//     PlcTask Inputs/GVL_iXlinker.EtherCAT_Master_EPPxxxx.Beckhoff_EPP3xxx.Beckhoff_EPP3xxxEK1122.A_0023_EPP3744_1041_0019.AI_Inputs_Channel_2.Value <-> AI Inputs Channel 2/Value
//     PlcTask Inputs/GVL_iXlinker.EtherCAT_Master_EPPxxxx.Beckhoff_EPP3xxx.Beckhoff_EPP3xxxEK1122.A_0023_EPP3744_1041_0019.AI_Inputs_Channel_3.Value <-> AI Inputs Channel 3/Value
//     PlcTask Inputs/GVL_iXlinker.EtherCAT_Master_EPPxxxx.Beckhoff_EPP3xxx.Beckhoff_EPP3xxxEK1122.A_0023_EPP3744_1041_0019.AI_Inputs_Channel_4.Value <-> AI Inputs Channel 4/Value
//     PlcTask Inputs/GVL_iXlinker.EtherCAT_Master_EPPxxxx.Beckhoff_EPP3xxx.Beckhoff_EPP3xxxEK1122.A_0023_EPP3744_1041_0019.DEV_Inputs_Device.Safe_State_Active <-> DEV Inputs Device/Safe State Active
//     PlcTask Inputs/GVL_iXlinker.EtherCAT_Master_EPPxxxx.Beckhoff_EPP3xxx.Beckhoff_EPP3xxxEK1122.A_0023_EPP3744_1041_0019.DEV_Inputs_Device.Sync_error <-> DEV Inputs Device/Sync error
//     PlcTask Inputs/GVL_iXlinker.EtherCAT_Master_EPPxxxx.Beckhoff_EPP3xxx.Beckhoff_EPP3xxxEK1122.A_0023_EPP3744_1041_0019.DEV_Inputs_Device.Undervoltage_Us <-> DEV Inputs Device/Undervoltage Us
//     PlcTask Inputs/GVL_iXlinker.EtherCAT_Master_EPPxxxx.Beckhoff_EPP3xxx.Beckhoff_EPP3xxxEK1122.A_0023_EPP3744_1041_0019.DEV_Inputs_Device.Undervoltage_Up <-> DEV Inputs Device/Undervoltage Up
//     PlcTask Inputs/GVL_iXlinker.EtherCAT_Master_EPPxxxx.Beckhoff_EPP3xxx.Beckhoff_EPP3xxxEK1122.A_0023_EPP3744_1041_0019.DEV_Inputs_Device.TxPDO_Toggle <-> DEV Inputs Device/TxPDO Toggle
//     PlcTask Outputs/GVL_iXlinker.EtherCAT_Master_EPPxxxx.Beckhoff_EPP3xxx.Beckhoff_EPP3xxxEK1122.A_0023_EPP3744_1041_0019.DIG_Outputs.Output[0] <-> DIG Outputs/Output 1
//     PlcTask Outputs/GVL_iXlinker.EtherCAT_Master_EPPxxxx.Beckhoff_EPP3xxx.Beckhoff_EPP3xxxEK1122.A_0023_EPP3744_1041_0019.DIG_Outputs.Output[1] <-> DIG Outputs/Output 2
//     PlcTask Outputs/GVL_iXlinker.EtherCAT_Master_EPPxxxx.Beckhoff_EPP3xxx.Beckhoff_EPP3xxxEK1122.A_0023_EPP3744_1041_0019.DEV_Outputs_Device.Set_safe_state <-> DEV Outputs Device/Set safe state
//     PlcTask Inputs/GVL_iXlinker.EtherCAT_Master_EPPxxxx.Beckhoff_EPP3xxx.Beckhoff_EPP3xxxEK1122.A_0023_EPP3744_1041_0019.WcState.WcState <-> WcState/WcState
//     PlcTask Inputs/GVL_iXlinker.EtherCAT_Master_EPPxxxx.Beckhoff_EPP3xxx.Beckhoff_EPP3xxxEK1122.A_0023_EPP3744_1041_0019.WcState.InputToggle <-> WcState/InputToggle
//     PlcTask Inputs/GVL_iXlinker.EtherCAT_Master_EPPxxxx.Beckhoff_EPP3xxx.Beckhoff_EPP3xxxEK1122.A_0023_EPP3744_1041_0019.InfoData.AdsAddr <-> InfoData/AdsAddr
//     PlcTask Inputs/GVL_iXlinker.EtherCAT_Master_EPPxxxx.Beckhoff_EPP3xxx.Beckhoff_EPP3xxxEK1122.A_0023_EPP3744_1041_0019.InfoData.State <-> InfoData/State
//   PLC/PLC Instance <-> EtherCAT Master EPPxxxx/Beckhoff EPP3xxx/Beckhoff EPP3xxxEK1122/A_0024(EPP3744-1041-0020)
//     PlcTask Inputs/GVL_iXlinker.EtherCAT_Master_EPPxxxx.Beckhoff_EPP3xxx.Beckhoff_EPP3xxxEK1122.A_0024_EPP3744_1041_0020.DIG_Inputs.Input[0] <-> DIG Inputs/Input 1
//     PlcTask Inputs/GVL_iXlinker.EtherCAT_Master_EPPxxxx.Beckhoff_EPP3xxx.Beckhoff_EPP3xxxEK1122.A_0024_EPP3744_1041_0020.DIG_Inputs.Input[1] <-> DIG Inputs/Input 2
//     PlcTask Inputs/GVL_iXlinker.EtherCAT_Master_EPPxxxx.Beckhoff_EPP3xxx.Beckhoff_EPP3xxxEK1122.A_0024_EPP3744_1041_0020.DIG_Inputs.Input[2] <-> DIG Inputs/Input 3
//     PlcTask Inputs/GVL_iXlinker.EtherCAT_Master_EPPxxxx.Beckhoff_EPP3xxx.Beckhoff_EPP3xxxEK1122.A_0024_EPP3744_1041_0020.DIG_Inputs.Input[3] <-> DIG Inputs/Input 4
//     PlcTask Inputs/GVL_iXlinker.EtherCAT_Master_EPPxxxx.Beckhoff_EPP3xxx.Beckhoff_EPP3xxxEK1122.A_0024_EPP3744_1041_0020.DIG_Inputs.Input[4] <-> DIG Inputs/Input 5
//     PlcTask Inputs/GVL_iXlinker.EtherCAT_Master_EPPxxxx.Beckhoff_EPP3xxx.Beckhoff_EPP3xxxEK1122.A_0024_EPP3744_1041_0020.DIG_Inputs.Input[5] <-> DIG Inputs/Input 6
//     PlcTask Inputs/GVL_iXlinker.EtherCAT_Master_EPPxxxx.Beckhoff_EPP3xxx.Beckhoff_EPP3xxxEK1122.A_0024_EPP3744_1041_0020.AI_Inputs_Channel_1.Status/Underrange <-> AI Inputs Channel 1/Status/Underrange
//     PlcTask Inputs/GVL_iXlinker.EtherCAT_Master_EPPxxxx.Beckhoff_EPP3xxx.Beckhoff_EPP3xxxEK1122.A_0024_EPP3744_1041_0020.AI_Inputs_Channel_2.Status/Underrange <-> AI Inputs Channel 2/Status/Underrange
//     PlcTask Inputs/GVL_iXlinker.EtherCAT_Master_EPPxxxx.Beckhoff_EPP3xxx.Beckhoff_EPP3xxxEK1122.A_0024_EPP3744_1041_0020.AI_Inputs_Channel_3.Status/Underrange <-> AI Inputs Channel 3/Status/Underrange
//     PlcTask Inputs/GVL_iXlinker.EtherCAT_Master_EPPxxxx.Beckhoff_EPP3xxx.Beckhoff_EPP3xxxEK1122.A_0024_EPP3744_1041_0020.AI_Inputs_Channel_4.Status/Underrange <-> AI Inputs Channel 4/Status/Underrange
//     PlcTask Inputs/GVL_iXlinker.EtherCAT_Master_EPPxxxx.Beckhoff_EPP3xxx.Beckhoff_EPP3xxxEK1122.A_0024_EPP3744_1041_0020.AI_Inputs_Channel_1.Status/Overrange <-> AI Inputs Channel 1/Status/Overrange
//     PlcTask Inputs/GVL_iXlinker.EtherCAT_Master_EPPxxxx.Beckhoff_EPP3xxx.Beckhoff_EPP3xxxEK1122.A_0024_EPP3744_1041_0020.AI_Inputs_Channel_2.Status/Overrange <-> AI Inputs Channel 2/Status/Overrange
//     PlcTask Inputs/GVL_iXlinker.EtherCAT_Master_EPPxxxx.Beckhoff_EPP3xxx.Beckhoff_EPP3xxxEK1122.A_0024_EPP3744_1041_0020.AI_Inputs_Channel_3.Status/Overrange <-> AI Inputs Channel 3/Status/Overrange
//     PlcTask Inputs/GVL_iXlinker.EtherCAT_Master_EPPxxxx.Beckhoff_EPP3xxx.Beckhoff_EPP3xxxEK1122.A_0024_EPP3744_1041_0020.AI_Inputs_Channel_4.Status/Overrange <-> AI Inputs Channel 4/Status/Overrange
//     PlcTask Inputs/GVL_iXlinker.EtherCAT_Master_EPPxxxx.Beckhoff_EPP3xxx.Beckhoff_EPP3xxxEK1122.A_0024_EPP3744_1041_0020.AI_Inputs_Channel_1.Status/Limit_1 <-> AI Inputs Channel 1/Status/Limit 1
//     PlcTask Inputs/GVL_iXlinker.EtherCAT_Master_EPPxxxx.Beckhoff_EPP3xxx.Beckhoff_EPP3xxxEK1122.A_0024_EPP3744_1041_0020.AI_Inputs_Channel_1.Status/Limit_2 <-> AI Inputs Channel 1/Status/Limit 2
//     PlcTask Inputs/GVL_iXlinker.EtherCAT_Master_EPPxxxx.Beckhoff_EPP3xxx.Beckhoff_EPP3xxxEK1122.A_0024_EPP3744_1041_0020.AI_Inputs_Channel_2.Status/Limit_1 <-> AI Inputs Channel 2/Status/Limit 1
//     PlcTask Inputs/GVL_iXlinker.EtherCAT_Master_EPPxxxx.Beckhoff_EPP3xxx.Beckhoff_EPP3xxxEK1122.A_0024_EPP3744_1041_0020.AI_Inputs_Channel_2.Status/Limit_2 <-> AI Inputs Channel 2/Status/Limit 2
//     PlcTask Inputs/GVL_iXlinker.EtherCAT_Master_EPPxxxx.Beckhoff_EPP3xxx.Beckhoff_EPP3xxxEK1122.A_0024_EPP3744_1041_0020.AI_Inputs_Channel_3.Status/Limit_1 <-> AI Inputs Channel 3/Status/Limit 1
//     PlcTask Inputs/GVL_iXlinker.EtherCAT_Master_EPPxxxx.Beckhoff_EPP3xxx.Beckhoff_EPP3xxxEK1122.A_0024_EPP3744_1041_0020.AI_Inputs_Channel_3.Status/Limit_2 <-> AI Inputs Channel 3/Status/Limit 2
//     PlcTask Inputs/GVL_iXlinker.EtherCAT_Master_EPPxxxx.Beckhoff_EPP3xxx.Beckhoff_EPP3xxxEK1122.A_0024_EPP3744_1041_0020.AI_Inputs_Channel_4.Status/Limit_1 <-> AI Inputs Channel 4/Status/Limit 1
//     PlcTask Inputs/GVL_iXlinker.EtherCAT_Master_EPPxxxx.Beckhoff_EPP3xxx.Beckhoff_EPP3xxxEK1122.A_0024_EPP3744_1041_0020.AI_Inputs_Channel_4.Status/Limit_2 <-> AI Inputs Channel 4/Status/Limit 2
//     PlcTask Inputs/GVL_iXlinker.EtherCAT_Master_EPPxxxx.Beckhoff_EPP3xxx.Beckhoff_EPP3xxxEK1122.A_0024_EPP3744_1041_0020.AI_Inputs_Channel_1.Status/Error <-> AI Inputs Channel 1/Status/Error
//     PlcTask Inputs/GVL_iXlinker.EtherCAT_Master_EPPxxxx.Beckhoff_EPP3xxx.Beckhoff_EPP3xxxEK1122.A_0024_EPP3744_1041_0020.AI_Inputs_Channel_2.Status/Error <-> AI Inputs Channel 2/Status/Error
//     PlcTask Inputs/GVL_iXlinker.EtherCAT_Master_EPPxxxx.Beckhoff_EPP3xxx.Beckhoff_EPP3xxxEK1122.A_0024_EPP3744_1041_0020.AI_Inputs_Channel_3.Status/Error <-> AI Inputs Channel 3/Status/Error
//     PlcTask Inputs/GVL_iXlinker.EtherCAT_Master_EPPxxxx.Beckhoff_EPP3xxx.Beckhoff_EPP3xxxEK1122.A_0024_EPP3744_1041_0020.AI_Inputs_Channel_4.Status/Error <-> AI Inputs Channel 4/Status/Error
//     PlcTask Inputs/GVL_iXlinker.EtherCAT_Master_EPPxxxx.Beckhoff_EPP3xxx.Beckhoff_EPP3xxxEK1122.A_0024_EPP3744_1041_0020.AI_Inputs_Channel_1.Status/TxPDO_State <-> AI Inputs Channel 1/Status/TxPDO State
//     PlcTask Inputs/GVL_iXlinker.EtherCAT_Master_EPPxxxx.Beckhoff_EPP3xxx.Beckhoff_EPP3xxxEK1122.A_0024_EPP3744_1041_0020.AI_Inputs_Channel_2.Status/TxPDO_State <-> AI Inputs Channel 2/Status/TxPDO State
//     PlcTask Inputs/GVL_iXlinker.EtherCAT_Master_EPPxxxx.Beckhoff_EPP3xxx.Beckhoff_EPP3xxxEK1122.A_0024_EPP3744_1041_0020.AI_Inputs_Channel_3.Status/TxPDO_State <-> AI Inputs Channel 3/Status/TxPDO State
//     PlcTask Inputs/GVL_iXlinker.EtherCAT_Master_EPPxxxx.Beckhoff_EPP3xxx.Beckhoff_EPP3xxxEK1122.A_0024_EPP3744_1041_0020.AI_Inputs_Channel_4.Status/TxPDO_State <-> AI Inputs Channel 4/Status/TxPDO State
//     PlcTask Inputs/GVL_iXlinker.EtherCAT_Master_EPPxxxx.Beckhoff_EPP3xxx.Beckhoff_EPP3xxxEK1122.A_0024_EPP3744_1041_0020.AI_Inputs_Channel_1.Status/TxPDO_Toggle <-> AI Inputs Channel 1/Status/TxPDO Toggle
//     PlcTask Inputs/GVL_iXlinker.EtherCAT_Master_EPPxxxx.Beckhoff_EPP3xxx.Beckhoff_EPP3xxxEK1122.A_0024_EPP3744_1041_0020.AI_Inputs_Channel_2.Status/TxPDO_Toggle <-> AI Inputs Channel 2/Status/TxPDO Toggle
//     PlcTask Inputs/GVL_iXlinker.EtherCAT_Master_EPPxxxx.Beckhoff_EPP3xxx.Beckhoff_EPP3xxxEK1122.A_0024_EPP3744_1041_0020.AI_Inputs_Channel_3.Status/TxPDO_Toggle <-> AI Inputs Channel 3/Status/TxPDO Toggle
//     PlcTask Inputs/GVL_iXlinker.EtherCAT_Master_EPPxxxx.Beckhoff_EPP3xxx.Beckhoff_EPP3xxxEK1122.A_0024_EPP3744_1041_0020.AI_Inputs_Channel_4.Status/TxPDO_Toggle <-> AI Inputs Channel 4/Status/TxPDO Toggle
//     PlcTask Inputs/GVL_iXlinker.EtherCAT_Master_EPPxxxx.Beckhoff_EPP3xxx.Beckhoff_EPP3xxxEK1122.A_0024_EPP3744_1041_0020.AI_Inputs_Channel_1.Value <-> AI Inputs Channel 1/Value
//     PlcTask Inputs/GVL_iXlinker.EtherCAT_Master_EPPxxxx.Beckhoff_EPP3xxx.Beckhoff_EPP3xxxEK1122.A_0024_EPP3744_1041_0020.AI_Inputs_Channel_2.Value <-> AI Inputs Channel 2/Value
//     PlcTask Inputs/GVL_iXlinker.EtherCAT_Master_EPPxxxx.Beckhoff_EPP3xxx.Beckhoff_EPP3xxxEK1122.A_0024_EPP3744_1041_0020.AI_Inputs_Channel_3.Value <-> AI Inputs Channel 3/Value
//     PlcTask Inputs/GVL_iXlinker.EtherCAT_Master_EPPxxxx.Beckhoff_EPP3xxx.Beckhoff_EPP3xxxEK1122.A_0024_EPP3744_1041_0020.AI_Inputs_Channel_4.Value <-> AI Inputs Channel 4/Value
//     PlcTask Inputs/GVL_iXlinker.EtherCAT_Master_EPPxxxx.Beckhoff_EPP3xxx.Beckhoff_EPP3xxxEK1122.A_0024_EPP3744_1041_0020.DEV_Inputs_Device.Safe_State_Active <-> DEV Inputs Device/Safe State Active
//     PlcTask Inputs/GVL_iXlinker.EtherCAT_Master_EPPxxxx.Beckhoff_EPP3xxx.Beckhoff_EPP3xxxEK1122.A_0024_EPP3744_1041_0020.DEV_Inputs_Device.Sync_error <-> DEV Inputs Device/Sync error
//     PlcTask Inputs/GVL_iXlinker.EtherCAT_Master_EPPxxxx.Beckhoff_EPP3xxx.Beckhoff_EPP3xxxEK1122.A_0024_EPP3744_1041_0020.DEV_Inputs_Device.Undervoltage_Us <-> DEV Inputs Device/Undervoltage Us
//     PlcTask Inputs/GVL_iXlinker.EtherCAT_Master_EPPxxxx.Beckhoff_EPP3xxx.Beckhoff_EPP3xxxEK1122.A_0024_EPP3744_1041_0020.DEV_Inputs_Device.Undervoltage_Up <-> DEV Inputs Device/Undervoltage Up
//     PlcTask Inputs/GVL_iXlinker.EtherCAT_Master_EPPxxxx.Beckhoff_EPP3xxx.Beckhoff_EPP3xxxEK1122.A_0024_EPP3744_1041_0020.DEV_Inputs_Device.TxPDO_Toggle <-> DEV Inputs Device/TxPDO Toggle
//     PlcTask Outputs/GVL_iXlinker.EtherCAT_Master_EPPxxxx.Beckhoff_EPP3xxx.Beckhoff_EPP3xxxEK1122.A_0024_EPP3744_1041_0020.DIG_Outputs.Output[0] <-> DIG Outputs/Output 1
//     PlcTask Outputs/GVL_iXlinker.EtherCAT_Master_EPPxxxx.Beckhoff_EPP3xxx.Beckhoff_EPP3xxxEK1122.A_0024_EPP3744_1041_0020.DIG_Outputs.Output[1] <-> DIG Outputs/Output 2
//     PlcTask Outputs/GVL_iXlinker.EtherCAT_Master_EPPxxxx.Beckhoff_EPP3xxx.Beckhoff_EPP3xxxEK1122.A_0024_EPP3744_1041_0020.DEV_Outputs_Device.Set_safe_state <-> DEV Outputs Device/Set safe state
//     PlcTask Inputs/GVL_iXlinker.EtherCAT_Master_EPPxxxx.Beckhoff_EPP3xxx.Beckhoff_EPP3xxxEK1122.A_0024_EPP3744_1041_0020.WcState.WcState <-> WcState/WcState
//     PlcTask Inputs/GVL_iXlinker.EtherCAT_Master_EPPxxxx.Beckhoff_EPP3xxx.Beckhoff_EPP3xxxEK1122.A_0024_EPP3744_1041_0020.WcState.InputToggle <-> WcState/InputToggle
//     PlcTask Inputs/GVL_iXlinker.EtherCAT_Master_EPPxxxx.Beckhoff_EPP3xxx.Beckhoff_EPP3xxxEK1122.A_0024_EPP3744_1041_0020.InfoData.AdsAddr <-> InfoData/AdsAddr
//     PlcTask Inputs/GVL_iXlinker.EtherCAT_Master_EPPxxxx.Beckhoff_EPP3xxx.Beckhoff_EPP3xxxEK1122.A_0024_EPP3744_1041_0020.InfoData.State <-> InfoData/State
//   PLC/PLC Instance <-> EtherCAT Master EPPxxxx/Beckhoff EPP3xxx/Beckhoff EPP3xxxEK1122/A_0025(EPP3752-0000-0017)
//     PlcTask Inputs/GVL_iXlinker.EtherCAT_Master_EPPxxxx.Beckhoff_EPP3xxx.Beckhoff_EPP3xxxEK1122.A_0025_EPP3752_0000_0017.AI_Inputs_Channel_1.Status/Error <-> AI Inputs Channel 1/Status/Error
//     PlcTask Inputs/GVL_iXlinker.EtherCAT_Master_EPPxxxx.Beckhoff_EPP3xxx.Beckhoff_EPP3xxxEK1122.A_0025_EPP3752_0000_0017.AI_Inputs_Channel_2.Status/Error <-> AI Inputs Channel 2/Status/Error
//     PlcTask Inputs/GVL_iXlinker.EtherCAT_Master_EPPxxxx.Beckhoff_EPP3xxx.Beckhoff_EPP3xxxEK1122.A_0025_EPP3752_0000_0017.AI_Inputs_Channel_3.Status/Error <-> AI Inputs Channel 3/Status/Error
//     PlcTask Inputs/GVL_iXlinker.EtherCAT_Master_EPPxxxx.Beckhoff_EPP3xxx.Beckhoff_EPP3xxxEK1122.A_0025_EPP3752_0000_0017.AI_Inputs_Channel_4.Status/Error <-> AI Inputs Channel 4/Status/Error
//     PlcTask Inputs/GVL_iXlinker.EtherCAT_Master_EPPxxxx.Beckhoff_EPP3xxx.Beckhoff_EPP3xxxEK1122.A_0025_EPP3752_0000_0017.AI_Inputs_Channel_5.Status/Error <-> AI Inputs Channel 5/Status/Error
//     PlcTask Inputs/GVL_iXlinker.EtherCAT_Master_EPPxxxx.Beckhoff_EPP3xxx.Beckhoff_EPP3xxxEK1122.A_0025_EPP3752_0000_0017.AI_Inputs_Channel_6.Status/Error <-> AI Inputs Channel 6/Status/Error
//     PlcTask Inputs/GVL_iXlinker.EtherCAT_Master_EPPxxxx.Beckhoff_EPP3xxx.Beckhoff_EPP3xxxEK1122.A_0025_EPP3752_0000_0017.AI_Inputs_Channel_1.Status/TxPDO_State <-> AI Inputs Channel 1/Status/TxPDO State
//     PlcTask Inputs/GVL_iXlinker.EtherCAT_Master_EPPxxxx.Beckhoff_EPP3xxx.Beckhoff_EPP3xxxEK1122.A_0025_EPP3752_0000_0017.AI_Inputs_Channel_2.Status/TxPDO_State <-> AI Inputs Channel 2/Status/TxPDO State
//     PlcTask Inputs/GVL_iXlinker.EtherCAT_Master_EPPxxxx.Beckhoff_EPP3xxx.Beckhoff_EPP3xxxEK1122.A_0025_EPP3752_0000_0017.AI_Inputs_Channel_3.Status/TxPDO_State <-> AI Inputs Channel 3/Status/TxPDO State
//     PlcTask Inputs/GVL_iXlinker.EtherCAT_Master_EPPxxxx.Beckhoff_EPP3xxx.Beckhoff_EPP3xxxEK1122.A_0025_EPP3752_0000_0017.AI_Inputs_Channel_4.Status/TxPDO_State <-> AI Inputs Channel 4/Status/TxPDO State
//     PlcTask Inputs/GVL_iXlinker.EtherCAT_Master_EPPxxxx.Beckhoff_EPP3xxx.Beckhoff_EPP3xxxEK1122.A_0025_EPP3752_0000_0017.AI_Inputs_Channel_5.Status/TxPDO_State <-> AI Inputs Channel 5/Status/TxPDO State
//     PlcTask Inputs/GVL_iXlinker.EtherCAT_Master_EPPxxxx.Beckhoff_EPP3xxx.Beckhoff_EPP3xxxEK1122.A_0025_EPP3752_0000_0017.AI_Inputs_Channel_6.Status/TxPDO_State <-> AI Inputs Channel 6/Status/TxPDO State
//     PlcTask Inputs/GVL_iXlinker.EtherCAT_Master_EPPxxxx.Beckhoff_EPP3xxx.Beckhoff_EPP3xxxEK1122.A_0025_EPP3752_0000_0017.AI_Inputs_Channel_1.Status/TxPDO_Toggle <-> AI Inputs Channel 1/Status/TxPDO Toggle
//     PlcTask Inputs/GVL_iXlinker.EtherCAT_Master_EPPxxxx.Beckhoff_EPP3xxx.Beckhoff_EPP3xxxEK1122.A_0025_EPP3752_0000_0017.AI_Inputs_Channel_2.Status/TxPDO_Toggle <-> AI Inputs Channel 2/Status/TxPDO Toggle
//     PlcTask Inputs/GVL_iXlinker.EtherCAT_Master_EPPxxxx.Beckhoff_EPP3xxx.Beckhoff_EPP3xxxEK1122.A_0025_EPP3752_0000_0017.AI_Inputs_Channel_3.Status/TxPDO_Toggle <-> AI Inputs Channel 3/Status/TxPDO Toggle
//     PlcTask Inputs/GVL_iXlinker.EtherCAT_Master_EPPxxxx.Beckhoff_EPP3xxx.Beckhoff_EPP3xxxEK1122.A_0025_EPP3752_0000_0017.AI_Inputs_Channel_4.Status/TxPDO_Toggle <-> AI Inputs Channel 4/Status/TxPDO Toggle
//     PlcTask Inputs/GVL_iXlinker.EtherCAT_Master_EPPxxxx.Beckhoff_EPP3xxx.Beckhoff_EPP3xxxEK1122.A_0025_EPP3752_0000_0017.AI_Inputs_Channel_5.Status/TxPDO_Toggle <-> AI Inputs Channel 5/Status/TxPDO Toggle
//     PlcTask Inputs/GVL_iXlinker.EtherCAT_Master_EPPxxxx.Beckhoff_EPP3xxx.Beckhoff_EPP3xxxEK1122.A_0025_EPP3752_0000_0017.AI_Inputs_Channel_6.Status/TxPDO_Toggle <-> AI Inputs Channel 6/Status/TxPDO Toggle
//     PlcTask Inputs/GVL_iXlinker.EtherCAT_Master_EPPxxxx.Beckhoff_EPP3xxx.Beckhoff_EPP3xxxEK1122.A_0025_EPP3752_0000_0017.AI_Inputs_Channel_1.Value <-> AI Inputs Channel 1/Value
//     PlcTask Inputs/GVL_iXlinker.EtherCAT_Master_EPPxxxx.Beckhoff_EPP3xxx.Beckhoff_EPP3xxxEK1122.A_0025_EPP3752_0000_0017.AI_Inputs_Channel_2.Value <-> AI Inputs Channel 2/Value
//     PlcTask Inputs/GVL_iXlinker.EtherCAT_Master_EPPxxxx.Beckhoff_EPP3xxx.Beckhoff_EPP3xxxEK1122.A_0025_EPP3752_0000_0017.AI_Inputs_Channel_3.Value <-> AI Inputs Channel 3/Value
//     PlcTask Inputs/GVL_iXlinker.EtherCAT_Master_EPPxxxx.Beckhoff_EPP3xxx.Beckhoff_EPP3xxxEK1122.A_0025_EPP3752_0000_0017.AI_Inputs_Channel_4.Value <-> AI Inputs Channel 4/Value
//     PlcTask Inputs/GVL_iXlinker.EtherCAT_Master_EPPxxxx.Beckhoff_EPP3xxx.Beckhoff_EPP3xxxEK1122.A_0025_EPP3752_0000_0017.AI_Inputs_Channel_5.Value <-> AI Inputs Channel 5/Value
//     PlcTask Inputs/GVL_iXlinker.EtherCAT_Master_EPPxxxx.Beckhoff_EPP3xxx.Beckhoff_EPP3xxxEK1122.A_0025_EPP3752_0000_0017.AI_Inputs_Channel_6.Value <-> AI Inputs Channel 6/Value
//     PlcTask Inputs/GVL_iXlinker.EtherCAT_Master_EPPxxxx.Beckhoff_EPP3xxx.Beckhoff_EPP3xxxEK1122.A_0025_EPP3752_0000_0017.WcState.WcState <-> WcState/WcState
//     PlcTask Inputs/GVL_iXlinker.EtherCAT_Master_EPPxxxx.Beckhoff_EPP3xxx.Beckhoff_EPP3xxxEK1122.A_0025_EPP3752_0000_0017.WcState.InputToggle <-> WcState/InputToggle
//     PlcTask Inputs/GVL_iXlinker.EtherCAT_Master_EPPxxxx.Beckhoff_EPP3xxx.Beckhoff_EPP3xxxEK1122.A_0025_EPP3752_0000_0017.InfoData.AdsAddr <-> InfoData/AdsAddr
//     PlcTask Inputs/GVL_iXlinker.EtherCAT_Master_EPPxxxx.Beckhoff_EPP3xxx.Beckhoff_EPP3xxxEK1122.A_0025_EPP3752_0000_0017.InfoData.State <-> InfoData/State
//   PLC/PLC Instance <-> EtherCAT Master EPPxxxx/Beckhoff EPP4xxx
//     PlcTask Inputs/GVL_iXlinker.EtherCAT_Master_EPPxxxx.Beckhoff_EPP4xxx.InfoData.State <-> InfoData/State
//   PLC/PLC Instance <-> EtherCAT Master EPPxxxx/Beckhoff EPP4xxx/Beckhoff EPP4xxxEK1122
//     PlcTask Inputs/GVL_iXlinker.EtherCAT_Master_EPPxxxx.Beckhoff_EPP4xxx.Beckhoff_EPP4xxxEK1122.InfoData.State <-> InfoData/State
//   PLC/PLC Instance <-> EtherCAT Master EPPxxxx/Beckhoff EPP4xxx/Beckhoff EPP4xxxEK1122/Beckhoff EPP4xxxsub EK1100
//     PlcTask Inputs/GVL_iXlinker.EtherCAT_Master_EPPxxxx.Beckhoff_EPP4xxx.Beckhoff_EPP4xxxEK1122.Beckhoff_EPP4xxxsub_EK1100.InfoData.State <-> InfoData/State
//   PLC/PLC Instance <-> EtherCAT Master EPPxxxx/Beckhoff EPP4xxx/Beckhoff EPP4xxxEK1122/A_0001(EPP4174-0002-0016)
//     PlcTask Outputs/GVL_iXlinker.EtherCAT_Master_EPPxxxx.Beckhoff_EPP4xxx.Beckhoff_EPP4xxxEK1122.A_0001_EPP4174_0002_0016.AO_Outputs_Channel_1.Analog_output <-> AO Outputs Channel 1/Analog output
//     PlcTask Outputs/GVL_iXlinker.EtherCAT_Master_EPPxxxx.Beckhoff_EPP4xxx.Beckhoff_EPP4xxxEK1122.A_0001_EPP4174_0002_0016.AO_Outputs_Channel_2.Analog_output <-> AO Outputs Channel 2/Analog output
//     PlcTask Outputs/GVL_iXlinker.EtherCAT_Master_EPPxxxx.Beckhoff_EPP4xxx.Beckhoff_EPP4xxxEK1122.A_0001_EPP4174_0002_0016.AO_Outputs_Channel_3.Analog_output <-> AO Outputs Channel 3/Analog output
//     PlcTask Outputs/GVL_iXlinker.EtherCAT_Master_EPPxxxx.Beckhoff_EPP4xxx.Beckhoff_EPP4xxxEK1122.A_0001_EPP4174_0002_0016.AO_Outputs_Channel_4.Analog_output <-> AO Outputs Channel 4/Analog output
//     PlcTask Inputs/GVL_iXlinker.EtherCAT_Master_EPPxxxx.Beckhoff_EPP4xxx.Beckhoff_EPP4xxxEK1122.A_0001_EPP4174_0002_0016.WcState.WcState <-> WcState/WcState
//     PlcTask Inputs/GVL_iXlinker.EtherCAT_Master_EPPxxxx.Beckhoff_EPP4xxx.Beckhoff_EPP4xxxEK1122.A_0001_EPP4174_0002_0016.InfoData.AdsAddr <-> InfoData/AdsAddr
//     PlcTask Inputs/GVL_iXlinker.EtherCAT_Master_EPPxxxx.Beckhoff_EPP4xxx.Beckhoff_EPP4xxxEK1122.A_0001_EPP4174_0002_0016.InfoData.State <-> InfoData/State
//   PLC/PLC Instance <-> EtherCAT Master EPPxxxx/Beckhoff EPP4xxx/Beckhoff EPP4xxxEK1122/A_0002(EPP4174-0002-0017)
//     PlcTask Outputs/GVL_iXlinker.EtherCAT_Master_EPPxxxx.Beckhoff_EPP4xxx.Beckhoff_EPP4xxxEK1122.A_0002_EPP4174_0002_0017.AO_Outputs_Channel_1.Analog_output <-> AO Outputs Channel 1/Analog output
//     PlcTask Outputs/GVL_iXlinker.EtherCAT_Master_EPPxxxx.Beckhoff_EPP4xxx.Beckhoff_EPP4xxxEK1122.A_0002_EPP4174_0002_0017.AO_Outputs_Channel_2.Analog_output <-> AO Outputs Channel 2/Analog output
//     PlcTask Outputs/GVL_iXlinker.EtherCAT_Master_EPPxxxx.Beckhoff_EPP4xxx.Beckhoff_EPP4xxxEK1122.A_0002_EPP4174_0002_0017.AO_Outputs_Channel_3.Analog_output <-> AO Outputs Channel 3/Analog output
//     PlcTask Outputs/GVL_iXlinker.EtherCAT_Master_EPPxxxx.Beckhoff_EPP4xxx.Beckhoff_EPP4xxxEK1122.A_0002_EPP4174_0002_0017.AO_Outputs_Channel_4.Analog_output <-> AO Outputs Channel 4/Analog output
//     PlcTask Inputs/GVL_iXlinker.EtherCAT_Master_EPPxxxx.Beckhoff_EPP4xxx.Beckhoff_EPP4xxxEK1122.A_0002_EPP4174_0002_0017.WcState.WcState <-> WcState/WcState
//     PlcTask Inputs/GVL_iXlinker.EtherCAT_Master_EPPxxxx.Beckhoff_EPP4xxx.Beckhoff_EPP4xxxEK1122.A_0002_EPP4174_0002_0017.InfoData.AdsAddr <-> InfoData/AdsAddr
//     PlcTask Inputs/GVL_iXlinker.EtherCAT_Master_EPPxxxx.Beckhoff_EPP4xxx.Beckhoff_EPP4xxxEK1122.A_0002_EPP4174_0002_0017.InfoData.State <-> InfoData/State
//   PLC/PLC Instance <-> EtherCAT Master EPPxxxx/Beckhoff EPP4xxx/Beckhoff EPP4xxxEK1122/A_0003(EPP4314-1002-0016)
//     PlcTask Inputs/GVL_iXlinker.EtherCAT_Master_EPPxxxx.Beckhoff_EPP4xxx.Beckhoff_EPP4xxxEK1122.A_0003_EPP4314_1002_0016.DI_Inputs.Input[0] <-> DI Inputs/Input 1
//     PlcTask Inputs/GVL_iXlinker.EtherCAT_Master_EPPxxxx.Beckhoff_EPP4xxx.Beckhoff_EPP4xxxEK1122.A_0003_EPP4314_1002_0016.DI_Inputs.Input[1] <-> DI Inputs/Input 2
//     PlcTask Inputs/GVL_iXlinker.EtherCAT_Master_EPPxxxx.Beckhoff_EPP4xxx.Beckhoff_EPP4xxxEK1122.A_0003_EPP4314_1002_0016.DI_Inputs.TxPDO_State <-> DI Inputs/TxPDO State
//     PlcTask Inputs/GVL_iXlinker.EtherCAT_Master_EPPxxxx.Beckhoff_EPP4xxx.Beckhoff_EPP4xxxEK1122.A_0003_EPP4314_1002_0016.DI_Inputs.TxPDO_Toggle <-> DI Inputs/TxPDO Toggle
//     PlcTask Inputs/GVL_iXlinker.EtherCAT_Master_EPPxxxx.Beckhoff_EPP4xxx.Beckhoff_EPP4xxxEK1122.A_0003_EPP4314_1002_0016.AI_Standard_Channel_1.Status/Underrange <-> AI Standard Channel 1/Status/Underrange
//     PlcTask Inputs/GVL_iXlinker.EtherCAT_Master_EPPxxxx.Beckhoff_EPP4xxx.Beckhoff_EPP4xxxEK1122.A_0003_EPP4314_1002_0016.AI_Standard_Channel_2.Status/Underrange <-> AI Standard Channel 2/Status/Underrange
//     PlcTask Inputs/GVL_iXlinker.EtherCAT_Master_EPPxxxx.Beckhoff_EPP4xxx.Beckhoff_EPP4xxxEK1122.A_0003_EPP4314_1002_0016.AI_Standard_Channel_1.Status/Overrange <-> AI Standard Channel 1/Status/Overrange
//     PlcTask Inputs/GVL_iXlinker.EtherCAT_Master_EPPxxxx.Beckhoff_EPP4xxx.Beckhoff_EPP4xxxEK1122.A_0003_EPP4314_1002_0016.AI_Standard_Channel_2.Status/Overrange <-> AI Standard Channel 2/Status/Overrange
//     PlcTask Inputs/GVL_iXlinker.EtherCAT_Master_EPPxxxx.Beckhoff_EPP4xxx.Beckhoff_EPP4xxxEK1122.A_0003_EPP4314_1002_0016.AI_Standard_Channel_1.Status/Limit_1 <-> AI Standard Channel 1/Status/Limit 1
//     PlcTask Inputs/GVL_iXlinker.EtherCAT_Master_EPPxxxx.Beckhoff_EPP4xxx.Beckhoff_EPP4xxxEK1122.A_0003_EPP4314_1002_0016.AI_Standard_Channel_1.Status/Limit_2 <-> AI Standard Channel 1/Status/Limit 2
//     PlcTask Inputs/GVL_iXlinker.EtherCAT_Master_EPPxxxx.Beckhoff_EPP4xxx.Beckhoff_EPP4xxxEK1122.A_0003_EPP4314_1002_0016.AI_Standard_Channel_2.Status/Limit_1 <-> AI Standard Channel 2/Status/Limit 1
//     PlcTask Inputs/GVL_iXlinker.EtherCAT_Master_EPPxxxx.Beckhoff_EPP4xxx.Beckhoff_EPP4xxxEK1122.A_0003_EPP4314_1002_0016.AI_Standard_Channel_2.Status/Limit_2 <-> AI Standard Channel 2/Status/Limit 2
//     PlcTask Inputs/GVL_iXlinker.EtherCAT_Master_EPPxxxx.Beckhoff_EPP4xxx.Beckhoff_EPP4xxxEK1122.A_0003_EPP4314_1002_0016.AI_Standard_Channel_1.Status/Error <-> AI Standard Channel 1/Status/Error
//     PlcTask Inputs/GVL_iXlinker.EtherCAT_Master_EPPxxxx.Beckhoff_EPP4xxx.Beckhoff_EPP4xxxEK1122.A_0003_EPP4314_1002_0016.AI_Standard_Channel_2.Status/Error <-> AI Standard Channel 2/Status/Error
//     PlcTask Inputs/GVL_iXlinker.EtherCAT_Master_EPPxxxx.Beckhoff_EPP4xxx.Beckhoff_EPP4xxxEK1122.A_0003_EPP4314_1002_0016.AI_Standard_Channel_1.Status/TxPDO_State <-> AI Standard Channel 1/Status/TxPDO State
//     PlcTask Inputs/GVL_iXlinker.EtherCAT_Master_EPPxxxx.Beckhoff_EPP4xxx.Beckhoff_EPP4xxxEK1122.A_0003_EPP4314_1002_0016.AI_Standard_Channel_2.Status/TxPDO_State <-> AI Standard Channel 2/Status/TxPDO State
//     PlcTask Inputs/GVL_iXlinker.EtherCAT_Master_EPPxxxx.Beckhoff_EPP4xxx.Beckhoff_EPP4xxxEK1122.A_0003_EPP4314_1002_0016.AI_Standard_Channel_1.Status/TxPDO_Toggle <-> AI Standard Channel 1/Status/TxPDO Toggle
//     PlcTask Inputs/GVL_iXlinker.EtherCAT_Master_EPPxxxx.Beckhoff_EPP4xxx.Beckhoff_EPP4xxxEK1122.A_0003_EPP4314_1002_0016.AI_Standard_Channel_2.Status/TxPDO_Toggle <-> AI Standard Channel 2/Status/TxPDO Toggle
//     PlcTask Inputs/GVL_iXlinker.EtherCAT_Master_EPPxxxx.Beckhoff_EPP4xxx.Beckhoff_EPP4xxxEK1122.A_0003_EPP4314_1002_0016.AI_Standard_Channel_1.Value <-> AI Standard Channel 1/Value
//     PlcTask Inputs/GVL_iXlinker.EtherCAT_Master_EPPxxxx.Beckhoff_EPP4xxx.Beckhoff_EPP4xxxEK1122.A_0003_EPP4314_1002_0016.AI_Standard_Channel_2.Value <-> AI Standard Channel 2/Value
//     PlcTask Outputs/GVL_iXlinker.EtherCAT_Master_EPPxxxx.Beckhoff_EPP4xxx.Beckhoff_EPP4xxxEK1122.A_0003_EPP4314_1002_0016.AO_Standard_Channel_1.Analog_output <-> AO Standard Channel 1/Analog output
//     PlcTask Outputs/GVL_iXlinker.EtherCAT_Master_EPPxxxx.Beckhoff_EPP4xxx.Beckhoff_EPP4xxxEK1122.A_0003_EPP4314_1002_0016.AO_Standard_Channel_2.Analog_output <-> AO Standard Channel 2/Analog output
//     PlcTask Inputs/GVL_iXlinker.EtherCAT_Master_EPPxxxx.Beckhoff_EPP4xxx.Beckhoff_EPP4xxxEK1122.A_0003_EPP4314_1002_0016.WcState.WcState <-> WcState/WcState
//     PlcTask Inputs/GVL_iXlinker.EtherCAT_Master_EPPxxxx.Beckhoff_EPP4xxx.Beckhoff_EPP4xxxEK1122.A_0003_EPP4314_1002_0016.WcState.InputToggle <-> WcState/InputToggle
//     PlcTask Inputs/GVL_iXlinker.EtherCAT_Master_EPPxxxx.Beckhoff_EPP4xxx.Beckhoff_EPP4xxxEK1122.A_0003_EPP4314_1002_0016.InfoData.AdsAddr <-> InfoData/AdsAddr
//     PlcTask Inputs/GVL_iXlinker.EtherCAT_Master_EPPxxxx.Beckhoff_EPP4xxx.Beckhoff_EPP4xxxEK1122.A_0003_EPP4314_1002_0016.InfoData.State <-> InfoData/State
//   PLC/PLC Instance <-> EtherCAT Master EPPxxxx/Beckhoff EPP4xxx/Beckhoff EPP4xxxEK1122/A_0004(EPP4374-0002-0016)
//     PlcTask Inputs/GVL_iXlinker.EtherCAT_Master_EPPxxxx.Beckhoff_EPP4xxx.Beckhoff_EPP4xxxEK1122.A_0004_EPP4374_0002_0016.AI_Inputs_Channel_1.Status/Underrange <-> AI Inputs Channel 1/Status/Underrange
//     PlcTask Inputs/GVL_iXlinker.EtherCAT_Master_EPPxxxx.Beckhoff_EPP4xxx.Beckhoff_EPP4xxxEK1122.A_0004_EPP4374_0002_0016.AI_Inputs_Channel_2.Status/Underrange <-> AI Inputs Channel 2/Status/Underrange
//     PlcTask Inputs/GVL_iXlinker.EtherCAT_Master_EPPxxxx.Beckhoff_EPP4xxx.Beckhoff_EPP4xxxEK1122.A_0004_EPP4374_0002_0016.AI_Inputs_Channel_1.Status/Overrange <-> AI Inputs Channel 1/Status/Overrange
//     PlcTask Inputs/GVL_iXlinker.EtherCAT_Master_EPPxxxx.Beckhoff_EPP4xxx.Beckhoff_EPP4xxxEK1122.A_0004_EPP4374_0002_0016.AI_Inputs_Channel_2.Status/Overrange <-> AI Inputs Channel 2/Status/Overrange
//     PlcTask Inputs/GVL_iXlinker.EtherCAT_Master_EPPxxxx.Beckhoff_EPP4xxx.Beckhoff_EPP4xxxEK1122.A_0004_EPP4374_0002_0016.AI_Inputs_Channel_1.Status/Limit_1 <-> AI Inputs Channel 1/Status/Limit 1
//     PlcTask Inputs/GVL_iXlinker.EtherCAT_Master_EPPxxxx.Beckhoff_EPP4xxx.Beckhoff_EPP4xxxEK1122.A_0004_EPP4374_0002_0016.AI_Inputs_Channel_1.Status/Limit_2 <-> AI Inputs Channel 1/Status/Limit 2
//     PlcTask Inputs/GVL_iXlinker.EtherCAT_Master_EPPxxxx.Beckhoff_EPP4xxx.Beckhoff_EPP4xxxEK1122.A_0004_EPP4374_0002_0016.AI_Inputs_Channel_2.Status/Limit_1 <-> AI Inputs Channel 2/Status/Limit 1
//     PlcTask Inputs/GVL_iXlinker.EtherCAT_Master_EPPxxxx.Beckhoff_EPP4xxx.Beckhoff_EPP4xxxEK1122.A_0004_EPP4374_0002_0016.AI_Inputs_Channel_2.Status/Limit_2 <-> AI Inputs Channel 2/Status/Limit 2
//     PlcTask Inputs/GVL_iXlinker.EtherCAT_Master_EPPxxxx.Beckhoff_EPP4xxx.Beckhoff_EPP4xxxEK1122.A_0004_EPP4374_0002_0016.AI_Inputs_Channel_1.Status/Error <-> AI Inputs Channel 1/Status/Error
//     PlcTask Inputs/GVL_iXlinker.EtherCAT_Master_EPPxxxx.Beckhoff_EPP4xxx.Beckhoff_EPP4xxxEK1122.A_0004_EPP4374_0002_0016.AI_Inputs_Channel_2.Status/Error <-> AI Inputs Channel 2/Status/Error
//     PlcTask Inputs/GVL_iXlinker.EtherCAT_Master_EPPxxxx.Beckhoff_EPP4xxx.Beckhoff_EPP4xxxEK1122.A_0004_EPP4374_0002_0016.AI_Inputs_Channel_1.Status/Sync_error <-> AI Inputs Channel 1/Status/Sync error
//     PlcTask Inputs/GVL_iXlinker.EtherCAT_Master_EPPxxxx.Beckhoff_EPP4xxx.Beckhoff_EPP4xxxEK1122.A_0004_EPP4374_0002_0016.AI_Inputs_Channel_2.Status/Sync_error <-> AI Inputs Channel 2/Status/Sync error
//     PlcTask Inputs/GVL_iXlinker.EtherCAT_Master_EPPxxxx.Beckhoff_EPP4xxx.Beckhoff_EPP4xxxEK1122.A_0004_EPP4374_0002_0016.AI_Inputs_Channel_1.Status/TxPDO_State <-> AI Inputs Channel 1/Status/TxPDO State
//     PlcTask Inputs/GVL_iXlinker.EtherCAT_Master_EPPxxxx.Beckhoff_EPP4xxx.Beckhoff_EPP4xxxEK1122.A_0004_EPP4374_0002_0016.AI_Inputs_Channel_2.Status/TxPDO_State <-> AI Inputs Channel 2/Status/TxPDO State
//     PlcTask Inputs/GVL_iXlinker.EtherCAT_Master_EPPxxxx.Beckhoff_EPP4xxx.Beckhoff_EPP4xxxEK1122.A_0004_EPP4374_0002_0016.AI_Inputs_Channel_1.Status/TxPDO_Toggle <-> AI Inputs Channel 1/Status/TxPDO Toggle
//     PlcTask Inputs/GVL_iXlinker.EtherCAT_Master_EPPxxxx.Beckhoff_EPP4xxx.Beckhoff_EPP4xxxEK1122.A_0004_EPP4374_0002_0016.AI_Inputs_Channel_2.Status/TxPDO_Toggle <-> AI Inputs Channel 2/Status/TxPDO Toggle
//     PlcTask Inputs/GVL_iXlinker.EtherCAT_Master_EPPxxxx.Beckhoff_EPP4xxx.Beckhoff_EPP4xxxEK1122.A_0004_EPP4374_0002_0016.AI_Inputs_Channel_1.Value <-> AI Inputs Channel 1/Value
//     PlcTask Inputs/GVL_iXlinker.EtherCAT_Master_EPPxxxx.Beckhoff_EPP4xxx.Beckhoff_EPP4xxxEK1122.A_0004_EPP4374_0002_0016.AI_Inputs_Channel_2.Value <-> AI Inputs Channel 2/Value
//     PlcTask Outputs/GVL_iXlinker.EtherCAT_Master_EPPxxxx.Beckhoff_EPP4xxx.Beckhoff_EPP4xxxEK1122.A_0004_EPP4374_0002_0016.AO_Outputs_Channel_3.Analog_output <-> AO Outputs Channel 3/Analog output
//     PlcTask Outputs/GVL_iXlinker.EtherCAT_Master_EPPxxxx.Beckhoff_EPP4xxx.Beckhoff_EPP4xxxEK1122.A_0004_EPP4374_0002_0016.AO_Outputs_Channel_4.Analog_output <-> AO Outputs Channel 4/Analog output
//     PlcTask Inputs/GVL_iXlinker.EtherCAT_Master_EPPxxxx.Beckhoff_EPP4xxx.Beckhoff_EPP4xxxEK1122.A_0004_EPP4374_0002_0016.WcState.WcState <-> WcState/WcState
//     PlcTask Inputs/GVL_iXlinker.EtherCAT_Master_EPPxxxx.Beckhoff_EPP4xxx.Beckhoff_EPP4xxxEK1122.A_0004_EPP4374_0002_0016.WcState.InputToggle <-> WcState/InputToggle
//     PlcTask Inputs/GVL_iXlinker.EtherCAT_Master_EPPxxxx.Beckhoff_EPP4xxx.Beckhoff_EPP4xxxEK1122.A_0004_EPP4374_0002_0016.InfoData.AdsAddr <-> InfoData/AdsAddr
//     PlcTask Inputs/GVL_iXlinker.EtherCAT_Master_EPPxxxx.Beckhoff_EPP4xxx.Beckhoff_EPP4xxxEK1122.A_0004_EPP4374_0002_0016.InfoData.State <-> InfoData/State
//   PLC/PLC Instance <-> EtherCAT Master EPPxxxx/Beckhoff EPP4xxx/Beckhoff EPP4xxxEK1122/A_0005(EPP4374-0002-0017)
//     PlcTask Inputs/GVL_iXlinker.EtherCAT_Master_EPPxxxx.Beckhoff_EPP4xxx.Beckhoff_EPP4xxxEK1122.A_0005_EPP4374_0002_0017.AI_Inputs_Channel_1.Status/Underrange <-> AI Inputs Channel 1/Status/Underrange
//     PlcTask Inputs/GVL_iXlinker.EtherCAT_Master_EPPxxxx.Beckhoff_EPP4xxx.Beckhoff_EPP4xxxEK1122.A_0005_EPP4374_0002_0017.AI_Inputs_Channel_2.Status/Underrange <-> AI Inputs Channel 2/Status/Underrange
//     PlcTask Inputs/GVL_iXlinker.EtherCAT_Master_EPPxxxx.Beckhoff_EPP4xxx.Beckhoff_EPP4xxxEK1122.A_0005_EPP4374_0002_0017.AI_Inputs_Channel_1.Status/Overrange <-> AI Inputs Channel 1/Status/Overrange
//     PlcTask Inputs/GVL_iXlinker.EtherCAT_Master_EPPxxxx.Beckhoff_EPP4xxx.Beckhoff_EPP4xxxEK1122.A_0005_EPP4374_0002_0017.AI_Inputs_Channel_2.Status/Overrange <-> AI Inputs Channel 2/Status/Overrange
//     PlcTask Inputs/GVL_iXlinker.EtherCAT_Master_EPPxxxx.Beckhoff_EPP4xxx.Beckhoff_EPP4xxxEK1122.A_0005_EPP4374_0002_0017.AI_Inputs_Channel_1.Status/Limit_1 <-> AI Inputs Channel 1/Status/Limit 1
//     PlcTask Inputs/GVL_iXlinker.EtherCAT_Master_EPPxxxx.Beckhoff_EPP4xxx.Beckhoff_EPP4xxxEK1122.A_0005_EPP4374_0002_0017.AI_Inputs_Channel_1.Status/Limit_2 <-> AI Inputs Channel 1/Status/Limit 2
//     PlcTask Inputs/GVL_iXlinker.EtherCAT_Master_EPPxxxx.Beckhoff_EPP4xxx.Beckhoff_EPP4xxxEK1122.A_0005_EPP4374_0002_0017.AI_Inputs_Channel_2.Status/Limit_1 <-> AI Inputs Channel 2/Status/Limit 1
//     PlcTask Inputs/GVL_iXlinker.EtherCAT_Master_EPPxxxx.Beckhoff_EPP4xxx.Beckhoff_EPP4xxxEK1122.A_0005_EPP4374_0002_0017.AI_Inputs_Channel_2.Status/Limit_2 <-> AI Inputs Channel 2/Status/Limit 2
//     PlcTask Inputs/GVL_iXlinker.EtherCAT_Master_EPPxxxx.Beckhoff_EPP4xxx.Beckhoff_EPP4xxxEK1122.A_0005_EPP4374_0002_0017.AI_Inputs_Channel_1.Status/Error <-> AI Inputs Channel 1/Status/Error
//     PlcTask Inputs/GVL_iXlinker.EtherCAT_Master_EPPxxxx.Beckhoff_EPP4xxx.Beckhoff_EPP4xxxEK1122.A_0005_EPP4374_0002_0017.AI_Inputs_Channel_2.Status/Error <-> AI Inputs Channel 2/Status/Error
//     PlcTask Inputs/GVL_iXlinker.EtherCAT_Master_EPPxxxx.Beckhoff_EPP4xxx.Beckhoff_EPP4xxxEK1122.A_0005_EPP4374_0002_0017.AI_Inputs_Channel_1.Status/Sync_error <-> AI Inputs Channel 1/Status/Sync error
//     PlcTask Inputs/GVL_iXlinker.EtherCAT_Master_EPPxxxx.Beckhoff_EPP4xxx.Beckhoff_EPP4xxxEK1122.A_0005_EPP4374_0002_0017.AI_Inputs_Channel_2.Status/Sync_error <-> AI Inputs Channel 2/Status/Sync error
//     PlcTask Inputs/GVL_iXlinker.EtherCAT_Master_EPPxxxx.Beckhoff_EPP4xxx.Beckhoff_EPP4xxxEK1122.A_0005_EPP4374_0002_0017.AI_Inputs_Channel_1.Status/TxPDO_State <-> AI Inputs Channel 1/Status/TxPDO State
//     PlcTask Inputs/GVL_iXlinker.EtherCAT_Master_EPPxxxx.Beckhoff_EPP4xxx.Beckhoff_EPP4xxxEK1122.A_0005_EPP4374_0002_0017.AI_Inputs_Channel_2.Status/TxPDO_State <-> AI Inputs Channel 2/Status/TxPDO State
//     PlcTask Inputs/GVL_iXlinker.EtherCAT_Master_EPPxxxx.Beckhoff_EPP4xxx.Beckhoff_EPP4xxxEK1122.A_0005_EPP4374_0002_0017.AI_Inputs_Channel_1.Status/TxPDO_Toggle <-> AI Inputs Channel 1/Status/TxPDO Toggle
//     PlcTask Inputs/GVL_iXlinker.EtherCAT_Master_EPPxxxx.Beckhoff_EPP4xxx.Beckhoff_EPP4xxxEK1122.A_0005_EPP4374_0002_0017.AI_Inputs_Channel_2.Status/TxPDO_Toggle <-> AI Inputs Channel 2/Status/TxPDO Toggle
//     PlcTask Inputs/GVL_iXlinker.EtherCAT_Master_EPPxxxx.Beckhoff_EPP4xxx.Beckhoff_EPP4xxxEK1122.A_0005_EPP4374_0002_0017.AI_Inputs_Channel_1.Value <-> AI Inputs Channel 1/Value
//     PlcTask Inputs/GVL_iXlinker.EtherCAT_Master_EPPxxxx.Beckhoff_EPP4xxx.Beckhoff_EPP4xxxEK1122.A_0005_EPP4374_0002_0017.AI_Inputs_Channel_2.Value <-> AI Inputs Channel 2/Value
//     PlcTask Outputs/GVL_iXlinker.EtherCAT_Master_EPPxxxx.Beckhoff_EPP4xxx.Beckhoff_EPP4xxxEK1122.A_0005_EPP4374_0002_0017.AO_Outputs_Channel_3.Analog_output <-> AO Outputs Channel 3/Analog output
//     PlcTask Outputs/GVL_iXlinker.EtherCAT_Master_EPPxxxx.Beckhoff_EPP4xxx.Beckhoff_EPP4xxxEK1122.A_0005_EPP4374_0002_0017.AO_Outputs_Channel_4.Analog_output <-> AO Outputs Channel 4/Analog output
//     PlcTask Inputs/GVL_iXlinker.EtherCAT_Master_EPPxxxx.Beckhoff_EPP4xxx.Beckhoff_EPP4xxxEK1122.A_0005_EPP4374_0002_0017.WcState.WcState <-> WcState/WcState
//     PlcTask Inputs/GVL_iXlinker.EtherCAT_Master_EPPxxxx.Beckhoff_EPP4xxx.Beckhoff_EPP4xxxEK1122.A_0005_EPP4374_0002_0017.WcState.InputToggle <-> WcState/InputToggle
//     PlcTask Inputs/GVL_iXlinker.EtherCAT_Master_EPPxxxx.Beckhoff_EPP4xxx.Beckhoff_EPP4xxxEK1122.A_0005_EPP4374_0002_0017.InfoData.AdsAddr <-> InfoData/AdsAddr
//     PlcTask Inputs/GVL_iXlinker.EtherCAT_Master_EPPxxxx.Beckhoff_EPP4xxx.Beckhoff_EPP4xxxEK1122.A_0005_EPP4374_0002_0017.InfoData.State <-> InfoData/State
//   PLC/PLC Instance <-> EtherCAT Master EPPxxxx/Beckhoff EPP4xxx/Beckhoff EPP4xxxEK1122/A_0006(EPP4374-0002-0018)
//     PlcTask Inputs/GVL_iXlinker.EtherCAT_Master_EPPxxxx.Beckhoff_EPP4xxx.Beckhoff_EPP4xxxEK1122.A_0006_EPP4374_0002_0018.AI_Inputs_Channel_1.Status/Underrange <-> AI Inputs Channel 1/Status/Underrange
//     PlcTask Inputs/GVL_iXlinker.EtherCAT_Master_EPPxxxx.Beckhoff_EPP4xxx.Beckhoff_EPP4xxxEK1122.A_0006_EPP4374_0002_0018.AI_Inputs_Channel_2.Status/Underrange <-> AI Inputs Channel 2/Status/Underrange
//     PlcTask Inputs/GVL_iXlinker.EtherCAT_Master_EPPxxxx.Beckhoff_EPP4xxx.Beckhoff_EPP4xxxEK1122.A_0006_EPP4374_0002_0018.AI_Inputs_Channel_1.Status/Overrange <-> AI Inputs Channel 1/Status/Overrange
//     PlcTask Inputs/GVL_iXlinker.EtherCAT_Master_EPPxxxx.Beckhoff_EPP4xxx.Beckhoff_EPP4xxxEK1122.A_0006_EPP4374_0002_0018.AI_Inputs_Channel_2.Status/Overrange <-> AI Inputs Channel 2/Status/Overrange
//     PlcTask Inputs/GVL_iXlinker.EtherCAT_Master_EPPxxxx.Beckhoff_EPP4xxx.Beckhoff_EPP4xxxEK1122.A_0006_EPP4374_0002_0018.AI_Inputs_Channel_1.Status/Limit_1 <-> AI Inputs Channel 1/Status/Limit 1
//     PlcTask Inputs/GVL_iXlinker.EtherCAT_Master_EPPxxxx.Beckhoff_EPP4xxx.Beckhoff_EPP4xxxEK1122.A_0006_EPP4374_0002_0018.AI_Inputs_Channel_1.Status/Limit_2 <-> AI Inputs Channel 1/Status/Limit 2
//     PlcTask Inputs/GVL_iXlinker.EtherCAT_Master_EPPxxxx.Beckhoff_EPP4xxx.Beckhoff_EPP4xxxEK1122.A_0006_EPP4374_0002_0018.AI_Inputs_Channel_2.Status/Limit_1 <-> AI Inputs Channel 2/Status/Limit 1
//     PlcTask Inputs/GVL_iXlinker.EtherCAT_Master_EPPxxxx.Beckhoff_EPP4xxx.Beckhoff_EPP4xxxEK1122.A_0006_EPP4374_0002_0018.AI_Inputs_Channel_2.Status/Limit_2 <-> AI Inputs Channel 2/Status/Limit 2
//     PlcTask Inputs/GVL_iXlinker.EtherCAT_Master_EPPxxxx.Beckhoff_EPP4xxx.Beckhoff_EPP4xxxEK1122.A_0006_EPP4374_0002_0018.AI_Inputs_Channel_1.Status/Error <-> AI Inputs Channel 1/Status/Error
//     PlcTask Inputs/GVL_iXlinker.EtherCAT_Master_EPPxxxx.Beckhoff_EPP4xxx.Beckhoff_EPP4xxxEK1122.A_0006_EPP4374_0002_0018.AI_Inputs_Channel_2.Status/Error <-> AI Inputs Channel 2/Status/Error
//     PlcTask Inputs/GVL_iXlinker.EtherCAT_Master_EPPxxxx.Beckhoff_EPP4xxx.Beckhoff_EPP4xxxEK1122.A_0006_EPP4374_0002_0018.AI_Inputs_Channel_1.Status/Sync_error <-> AI Inputs Channel 1/Status/Sync error
//     PlcTask Inputs/GVL_iXlinker.EtherCAT_Master_EPPxxxx.Beckhoff_EPP4xxx.Beckhoff_EPP4xxxEK1122.A_0006_EPP4374_0002_0018.AI_Inputs_Channel_2.Status/Sync_error <-> AI Inputs Channel 2/Status/Sync error
//     PlcTask Inputs/GVL_iXlinker.EtherCAT_Master_EPPxxxx.Beckhoff_EPP4xxx.Beckhoff_EPP4xxxEK1122.A_0006_EPP4374_0002_0018.AI_Inputs_Channel_1.Status/TxPDO_State <-> AI Inputs Channel 1/Status/TxPDO State
//     PlcTask Inputs/GVL_iXlinker.EtherCAT_Master_EPPxxxx.Beckhoff_EPP4xxx.Beckhoff_EPP4xxxEK1122.A_0006_EPP4374_0002_0018.AI_Inputs_Channel_2.Status/TxPDO_State <-> AI Inputs Channel 2/Status/TxPDO State
//     PlcTask Inputs/GVL_iXlinker.EtherCAT_Master_EPPxxxx.Beckhoff_EPP4xxx.Beckhoff_EPP4xxxEK1122.A_0006_EPP4374_0002_0018.AI_Inputs_Channel_1.Status/TxPDO_Toggle <-> AI Inputs Channel 1/Status/TxPDO Toggle
//     PlcTask Inputs/GVL_iXlinker.EtherCAT_Master_EPPxxxx.Beckhoff_EPP4xxx.Beckhoff_EPP4xxxEK1122.A_0006_EPP4374_0002_0018.AI_Inputs_Channel_2.Status/TxPDO_Toggle <-> AI Inputs Channel 2/Status/TxPDO Toggle
//     PlcTask Inputs/GVL_iXlinker.EtherCAT_Master_EPPxxxx.Beckhoff_EPP4xxx.Beckhoff_EPP4xxxEK1122.A_0006_EPP4374_0002_0018.AI_Inputs_Channel_1.Value <-> AI Inputs Channel 1/Value
//     PlcTask Inputs/GVL_iXlinker.EtherCAT_Master_EPPxxxx.Beckhoff_EPP4xxx.Beckhoff_EPP4xxxEK1122.A_0006_EPP4374_0002_0018.AI_Inputs_Channel_2.Value <-> AI Inputs Channel 2/Value
//     PlcTask Outputs/GVL_iXlinker.EtherCAT_Master_EPPxxxx.Beckhoff_EPP4xxx.Beckhoff_EPP4xxxEK1122.A_0006_EPP4374_0002_0018.AO_Outputs_Channel_3.Analog_output <-> AO Outputs Channel 3/Analog output
//     PlcTask Outputs/GVL_iXlinker.EtherCAT_Master_EPPxxxx.Beckhoff_EPP4xxx.Beckhoff_EPP4xxxEK1122.A_0006_EPP4374_0002_0018.AO_Outputs_Channel_4.Analog_output <-> AO Outputs Channel 4/Analog output
//     PlcTask Inputs/GVL_iXlinker.EtherCAT_Master_EPPxxxx.Beckhoff_EPP4xxx.Beckhoff_EPP4xxxEK1122.A_0006_EPP4374_0002_0018.WcState.WcState <-> WcState/WcState
//     PlcTask Inputs/GVL_iXlinker.EtherCAT_Master_EPPxxxx.Beckhoff_EPP4xxx.Beckhoff_EPP4xxxEK1122.A_0006_EPP4374_0002_0018.WcState.InputToggle <-> WcState/InputToggle
//     PlcTask Inputs/GVL_iXlinker.EtherCAT_Master_EPPxxxx.Beckhoff_EPP4xxx.Beckhoff_EPP4xxxEK1122.A_0006_EPP4374_0002_0018.InfoData.AdsAddr <-> InfoData/AdsAddr
//     PlcTask Inputs/GVL_iXlinker.EtherCAT_Master_EPPxxxx.Beckhoff_EPP4xxx.Beckhoff_EPP4xxxEK1122.A_0006_EPP4374_0002_0018.InfoData.State <-> InfoData/State
//   PLC/PLC Instance <-> EtherCAT Master EPPxxxx/Beckhoff EPP4xxx/Beckhoff EPP4xxxEK1122/A_0007(EPP4374-0002-0019)
//     PlcTask Inputs/GVL_iXlinker.EtherCAT_Master_EPPxxxx.Beckhoff_EPP4xxx.Beckhoff_EPP4xxxEK1122.A_0007_EPP4374_0002_0019.AI_Inputs_Channel_1.Status/Underrange <-> AI Inputs Channel 1/Status/Underrange
//     PlcTask Inputs/GVL_iXlinker.EtherCAT_Master_EPPxxxx.Beckhoff_EPP4xxx.Beckhoff_EPP4xxxEK1122.A_0007_EPP4374_0002_0019.AI_Inputs_Channel_2.Status/Underrange <-> AI Inputs Channel 2/Status/Underrange
//     PlcTask Inputs/GVL_iXlinker.EtherCAT_Master_EPPxxxx.Beckhoff_EPP4xxx.Beckhoff_EPP4xxxEK1122.A_0007_EPP4374_0002_0019.AI_Inputs_Channel_1.Status/Overrange <-> AI Inputs Channel 1/Status/Overrange
//     PlcTask Inputs/GVL_iXlinker.EtherCAT_Master_EPPxxxx.Beckhoff_EPP4xxx.Beckhoff_EPP4xxxEK1122.A_0007_EPP4374_0002_0019.AI_Inputs_Channel_2.Status/Overrange <-> AI Inputs Channel 2/Status/Overrange
//     PlcTask Inputs/GVL_iXlinker.EtherCAT_Master_EPPxxxx.Beckhoff_EPP4xxx.Beckhoff_EPP4xxxEK1122.A_0007_EPP4374_0002_0019.AI_Inputs_Channel_1.Status/Limit_1 <-> AI Inputs Channel 1/Status/Limit 1
//     PlcTask Inputs/GVL_iXlinker.EtherCAT_Master_EPPxxxx.Beckhoff_EPP4xxx.Beckhoff_EPP4xxxEK1122.A_0007_EPP4374_0002_0019.AI_Inputs_Channel_1.Status/Limit_2 <-> AI Inputs Channel 1/Status/Limit 2
//     PlcTask Inputs/GVL_iXlinker.EtherCAT_Master_EPPxxxx.Beckhoff_EPP4xxx.Beckhoff_EPP4xxxEK1122.A_0007_EPP4374_0002_0019.AI_Inputs_Channel_2.Status/Limit_1 <-> AI Inputs Channel 2/Status/Limit 1
//     PlcTask Inputs/GVL_iXlinker.EtherCAT_Master_EPPxxxx.Beckhoff_EPP4xxx.Beckhoff_EPP4xxxEK1122.A_0007_EPP4374_0002_0019.AI_Inputs_Channel_2.Status/Limit_2 <-> AI Inputs Channel 2/Status/Limit 2
//     PlcTask Inputs/GVL_iXlinker.EtherCAT_Master_EPPxxxx.Beckhoff_EPP4xxx.Beckhoff_EPP4xxxEK1122.A_0007_EPP4374_0002_0019.AI_Inputs_Channel_1.Status/Error <-> AI Inputs Channel 1/Status/Error
//     PlcTask Inputs/GVL_iXlinker.EtherCAT_Master_EPPxxxx.Beckhoff_EPP4xxx.Beckhoff_EPP4xxxEK1122.A_0007_EPP4374_0002_0019.AI_Inputs_Channel_2.Status/Error <-> AI Inputs Channel 2/Status/Error
//     PlcTask Inputs/GVL_iXlinker.EtherCAT_Master_EPPxxxx.Beckhoff_EPP4xxx.Beckhoff_EPP4xxxEK1122.A_0007_EPP4374_0002_0019.AI_Inputs_Channel_1.Status/Sync_error <-> AI Inputs Channel 1/Status/Sync error
//     PlcTask Inputs/GVL_iXlinker.EtherCAT_Master_EPPxxxx.Beckhoff_EPP4xxx.Beckhoff_EPP4xxxEK1122.A_0007_EPP4374_0002_0019.AI_Inputs_Channel_2.Status/Sync_error <-> AI Inputs Channel 2/Status/Sync error
//     PlcTask Inputs/GVL_iXlinker.EtherCAT_Master_EPPxxxx.Beckhoff_EPP4xxx.Beckhoff_EPP4xxxEK1122.A_0007_EPP4374_0002_0019.AI_Inputs_Channel_1.Status/TxPDO_State <-> AI Inputs Channel 1/Status/TxPDO State
//     PlcTask Inputs/GVL_iXlinker.EtherCAT_Master_EPPxxxx.Beckhoff_EPP4xxx.Beckhoff_EPP4xxxEK1122.A_0007_EPP4374_0002_0019.AI_Inputs_Channel_2.Status/TxPDO_State <-> AI Inputs Channel 2/Status/TxPDO State
//     PlcTask Inputs/GVL_iXlinker.EtherCAT_Master_EPPxxxx.Beckhoff_EPP4xxx.Beckhoff_EPP4xxxEK1122.A_0007_EPP4374_0002_0019.AI_Inputs_Channel_1.Status/TxPDO_Toggle <-> AI Inputs Channel 1/Status/TxPDO Toggle
//     PlcTask Inputs/GVL_iXlinker.EtherCAT_Master_EPPxxxx.Beckhoff_EPP4xxx.Beckhoff_EPP4xxxEK1122.A_0007_EPP4374_0002_0019.AI_Inputs_Channel_2.Status/TxPDO_Toggle <-> AI Inputs Channel 2/Status/TxPDO Toggle
//     PlcTask Inputs/GVL_iXlinker.EtherCAT_Master_EPPxxxx.Beckhoff_EPP4xxx.Beckhoff_EPP4xxxEK1122.A_0007_EPP4374_0002_0019.AI_Inputs_Channel_1.Value <-> AI Inputs Channel 1/Value
//     PlcTask Inputs/GVL_iXlinker.EtherCAT_Master_EPPxxxx.Beckhoff_EPP4xxx.Beckhoff_EPP4xxxEK1122.A_0007_EPP4374_0002_0019.AI_Inputs_Channel_2.Value <-> AI Inputs Channel 2/Value
//     PlcTask Outputs/GVL_iXlinker.EtherCAT_Master_EPPxxxx.Beckhoff_EPP4xxx.Beckhoff_EPP4xxxEK1122.A_0007_EPP4374_0002_0019.AO_Outputs_Channel_3.Analog_output <-> AO Outputs Channel 3/Analog output
//     PlcTask Outputs/GVL_iXlinker.EtherCAT_Master_EPPxxxx.Beckhoff_EPP4xxx.Beckhoff_EPP4xxxEK1122.A_0007_EPP4374_0002_0019.AO_Outputs_Channel_4.Analog_output <-> AO Outputs Channel 4/Analog output
//     PlcTask Inputs/GVL_iXlinker.EtherCAT_Master_EPPxxxx.Beckhoff_EPP4xxx.Beckhoff_EPP4xxxEK1122.A_0007_EPP4374_0002_0019.WcState.WcState <-> WcState/WcState
//     PlcTask Inputs/GVL_iXlinker.EtherCAT_Master_EPPxxxx.Beckhoff_EPP4xxx.Beckhoff_EPP4xxxEK1122.A_0007_EPP4374_0002_0019.WcState.InputToggle <-> WcState/InputToggle
//     PlcTask Inputs/GVL_iXlinker.EtherCAT_Master_EPPxxxx.Beckhoff_EPP4xxx.Beckhoff_EPP4xxxEK1122.A_0007_EPP4374_0002_0019.InfoData.AdsAddr <-> InfoData/AdsAddr
//     PlcTask Inputs/GVL_iXlinker.EtherCAT_Master_EPPxxxx.Beckhoff_EPP4xxx.Beckhoff_EPP4xxxEK1122.A_0007_EPP4374_0002_0019.InfoData.State <-> InfoData/State
//   PLC/PLC Instance <-> EtherCAT Master EPPxxxx/Beckhoff EPP5xxx
//     PlcTask Inputs/GVL_iXlinker.EtherCAT_Master_EPPxxxx.Beckhoff_EPP5xxx.InfoData.State <-> InfoData/State
//   PLC/PLC Instance <-> EtherCAT Master EPPxxxx/Beckhoff EPP5xxx/Beckhoff EPP5xxxEK1122
//     PlcTask Inputs/GVL_iXlinker.EtherCAT_Master_EPPxxxx.Beckhoff_EPP5xxx.Beckhoff_EPP5xxxEK1122.InfoData.State <-> InfoData/State
//   PLC/PLC Instance <-> EtherCAT Master EPPxxxx/Beckhoff EPP5xxx/Beckhoff EPP5xxxEK1122/Beckhoff EPP5xxxsub EK1100
//     PlcTask Inputs/GVL_iXlinker.EtherCAT_Master_EPPxxxx.Beckhoff_EPP5xxx.Beckhoff_EPP5xxxEK1122.Beckhoff_EPP5xxxsub_EK1100.InfoData.State <-> InfoData/State
//   PLC/PLC Instance <-> EtherCAT Master EPPxxxx/Beckhoff EPP5xxx/Beckhoff EPP5xxxEK1122/A_0001(EPP5001-0002-0016)
//     PlcTask Inputs/GVL_iXlinker.EtherCAT_Master_EPPxxxx.Beckhoff_EPP5xxx.Beckhoff_EPP5xxxEK1122.A_0001_EPP5001_0002_0016.SSI_Inputs.Status/Data_error <-> SSI Inputs/Status/Data error
//     PlcTask Inputs/GVL_iXlinker.EtherCAT_Master_EPPxxxx.Beckhoff_EPP5xxx.Beckhoff_EPP5xxxEK1122.A_0001_EPP5001_0002_0016.SSI_Inputs.Status/Frame_error <-> SSI Inputs/Status/Frame error
//     PlcTask Inputs/GVL_iXlinker.EtherCAT_Master_EPPxxxx.Beckhoff_EPP5xxx.Beckhoff_EPP5xxxEK1122.A_0001_EPP5001_0002_0016.SSI_Inputs.Status/Power_failure <-> SSI Inputs/Status/Power failure
//     PlcTask Inputs/GVL_iXlinker.EtherCAT_Master_EPPxxxx.Beckhoff_EPP5xxx.Beckhoff_EPP5xxxEK1122.A_0001_EPP5001_0002_0016.SSI_Inputs.Status/Sync_error <-> SSI Inputs/Status/Sync error
//     PlcTask Inputs/GVL_iXlinker.EtherCAT_Master_EPPxxxx.Beckhoff_EPP5xxx.Beckhoff_EPP5xxxEK1122.A_0001_EPP5001_0002_0016.SSI_Inputs.Status/TxPDO_State <-> SSI Inputs/Status/TxPDO State
//     PlcTask Inputs/GVL_iXlinker.EtherCAT_Master_EPPxxxx.Beckhoff_EPP5xxx.Beckhoff_EPP5xxxEK1122.A_0001_EPP5001_0002_0016.SSI_Inputs.Status/TxPDO_Toggle <-> SSI Inputs/Status/TxPDO Toggle
//     PlcTask Inputs/GVL_iXlinker.EtherCAT_Master_EPPxxxx.Beckhoff_EPP5xxx.Beckhoff_EPP5xxxEK1122.A_0001_EPP5001_0002_0016.SSI_Inputs.Counter_value <-> SSI Inputs/Counter value
//     PlcTask Inputs/GVL_iXlinker.EtherCAT_Master_EPPxxxx.Beckhoff_EPP5xxx.Beckhoff_EPP5xxxEK1122.A_0001_EPP5001_0002_0016.WcState.WcState <-> WcState/WcState
//     PlcTask Inputs/GVL_iXlinker.EtherCAT_Master_EPPxxxx.Beckhoff_EPP5xxx.Beckhoff_EPP5xxxEK1122.A_0001_EPP5001_0002_0016.WcState.InputToggle <-> WcState/InputToggle
//     PlcTask Inputs/GVL_iXlinker.EtherCAT_Master_EPPxxxx.Beckhoff_EPP5xxx.Beckhoff_EPP5xxxEK1122.A_0001_EPP5001_0002_0016.InfoData.AdsAddr <-> InfoData/AdsAddr
//     PlcTask Inputs/GVL_iXlinker.EtherCAT_Master_EPPxxxx.Beckhoff_EPP5xxx.Beckhoff_EPP5xxxEK1122.A_0001_EPP5001_0002_0016.InfoData.State <-> InfoData/State
//   PLC/PLC Instance <-> EtherCAT Master EPPxxxx/Beckhoff EPP5xxx/Beckhoff EPP5xxxEK1122/A_0002(EPP5101-0002-0016)
//     PlcTask Inputs/GVL_iXlinker.EtherCAT_Master_EPPxxxx.Beckhoff_EPP5xxx.Beckhoff_EPP5xxxEK1122.A_0002_EPP5101_0002_0016.ENC_Status_compact.Status/Latch_C_valid <-> ENC Status compact/Status/Latch C valid
//     PlcTask Inputs/GVL_iXlinker.EtherCAT_Master_EPPxxxx.Beckhoff_EPP5xxx.Beckhoff_EPP5xxxEK1122.A_0002_EPP5101_0002_0016.ENC_Status_compact.Status/Set_counter_done <-> ENC Status compact/Status/Set counter done
//     PlcTask Inputs/GVL_iXlinker.EtherCAT_Master_EPPxxxx.Beckhoff_EPP5xxx.Beckhoff_EPP5xxxEK1122.A_0002_EPP5101_0002_0016.ENC_Status_compact.Status/Counter_underflow <-> ENC Status compact/Status/Counter underflow
//     PlcTask Inputs/GVL_iXlinker.EtherCAT_Master_EPPxxxx.Beckhoff_EPP5xxx.Beckhoff_EPP5xxxEK1122.A_0002_EPP5101_0002_0016.ENC_Status_compact.Status/Counter_overflow <-> ENC Status compact/Status/Counter overflow
//     PlcTask Inputs/GVL_iXlinker.EtherCAT_Master_EPPxxxx.Beckhoff_EPP5xxx.Beckhoff_EPP5xxxEK1122.A_0002_EPP5101_0002_0016.ENC_Status_compact.Status/Open_circuit <-> ENC Status compact/Status/Open circuit
//     PlcTask Inputs/GVL_iXlinker.EtherCAT_Master_EPPxxxx.Beckhoff_EPP5xxx.Beckhoff_EPP5xxxEK1122.A_0002_EPP5101_0002_0016.ENC_Status_compact.Status/Extrapolation_stall <-> ENC Status compact/Status/Extrapolation stall
//     PlcTask Inputs/GVL_iXlinker.EtherCAT_Master_EPPxxxx.Beckhoff_EPP5xxx.Beckhoff_EPP5xxxEK1122.A_0002_EPP5101_0002_0016.ENC_Status_compact.Status/Status_of_input_A <-> ENC Status compact/Status/Status of input A
//     PlcTask Inputs/GVL_iXlinker.EtherCAT_Master_EPPxxxx.Beckhoff_EPP5xxx.Beckhoff_EPP5xxxEK1122.A_0002_EPP5101_0002_0016.ENC_Status_compact.Status/Status_of_input_B <-> ENC Status compact/Status/Status of input B
//     PlcTask Inputs/GVL_iXlinker.EtherCAT_Master_EPPxxxx.Beckhoff_EPP5xxx.Beckhoff_EPP5xxxEK1122.A_0002_EPP5101_0002_0016.ENC_Status_compact.Status/Status_of_input_C <-> ENC Status compact/Status/Status of input C
//     PlcTask Inputs/GVL_iXlinker.EtherCAT_Master_EPPxxxx.Beckhoff_EPP5xxx.Beckhoff_EPP5xxxEK1122.A_0002_EPP5101_0002_0016.ENC_Status_compact.Status/Sync_error <-> ENC Status compact/Status/Sync error
//     PlcTask Inputs/GVL_iXlinker.EtherCAT_Master_EPPxxxx.Beckhoff_EPP5xxx.Beckhoff_EPP5xxxEK1122.A_0002_EPP5101_0002_0016.ENC_Status_compact.Status/TxPDO_State <-> ENC Status compact/Status/TxPDO State
//     PlcTask Inputs/GVL_iXlinker.EtherCAT_Master_EPPxxxx.Beckhoff_EPP5xxx.Beckhoff_EPP5xxxEK1122.A_0002_EPP5101_0002_0016.ENC_Status_compact.Status/TxPDO_Toggle <-> ENC Status compact/Status/TxPDO Toggle
//     PlcTask Inputs/GVL_iXlinker.EtherCAT_Master_EPPxxxx.Beckhoff_EPP5xxx.Beckhoff_EPP5xxxEK1122.A_0002_EPP5101_0002_0016.ENC_Status_compact.Counter_value <-> ENC Status compact/Counter value
//     PlcTask Inputs/GVL_iXlinker.EtherCAT_Master_EPPxxxx.Beckhoff_EPP5xxx.Beckhoff_EPP5xxxEK1122.A_0002_EPP5101_0002_0016.ENC_Status_compact.Latch_value <-> ENC Status compact/Latch value
//     PlcTask Outputs/GVL_iXlinker.EtherCAT_Master_EPPxxxx.Beckhoff_EPP5xxx.Beckhoff_EPP5xxxEK1122.A_0002_EPP5101_0002_0016.ENC_Control_compact.Control/Enable_latch_C <-> ENC Control compact/Control/Enable latch C
//     PlcTask Outputs/GVL_iXlinker.EtherCAT_Master_EPPxxxx.Beckhoff_EPP5xxx.Beckhoff_EPP5xxxEK1122.A_0002_EPP5101_0002_0016.ENC_Control_compact.Control/Set_counter <-> ENC Control compact/Control/Set counter
//     PlcTask Outputs/GVL_iXlinker.EtherCAT_Master_EPPxxxx.Beckhoff_EPP5xxx.Beckhoff_EPP5xxxEK1122.A_0002_EPP5101_0002_0016.ENC_Control_compact.Set_counter_value <-> ENC Control compact/Set counter value
//     PlcTask Inputs/GVL_iXlinker.EtherCAT_Master_EPPxxxx.Beckhoff_EPP5xxx.Beckhoff_EPP5xxxEK1122.A_0002_EPP5101_0002_0016.WcState.WcState <-> WcState/WcState
//     PlcTask Inputs/GVL_iXlinker.EtherCAT_Master_EPPxxxx.Beckhoff_EPP5xxx.Beckhoff_EPP5xxxEK1122.A_0002_EPP5101_0002_0016.WcState.InputToggle <-> WcState/InputToggle
//     PlcTask Inputs/GVL_iXlinker.EtherCAT_Master_EPPxxxx.Beckhoff_EPP5xxx.Beckhoff_EPP5xxxEK1122.A_0002_EPP5101_0002_0016.InfoData.AdsAddr <-> InfoData/AdsAddr
//     PlcTask Inputs/GVL_iXlinker.EtherCAT_Master_EPPxxxx.Beckhoff_EPP5xxx.Beckhoff_EPP5xxxEK1122.A_0002_EPP5101_0002_0016.InfoData.State <-> InfoData/State
//   PLC/PLC Instance <-> EtherCAT Master EPPxxxx/Beckhoff EPP5xxx/Beckhoff EPP5xxxEK1122/A_0003(EPP5101-0002-0017)
//     PlcTask Inputs/GVL_iXlinker.EtherCAT_Master_EPPxxxx.Beckhoff_EPP5xxx.Beckhoff_EPP5xxxEK1122.A_0003_EPP5101_0002_0017.ENC_Status_compact.Status/Latch_C_valid <-> ENC Status compact/Status/Latch C valid
//     PlcTask Inputs/GVL_iXlinker.EtherCAT_Master_EPPxxxx.Beckhoff_EPP5xxx.Beckhoff_EPP5xxxEK1122.A_0003_EPP5101_0002_0017.ENC_Status_compact.Status/Set_counter_done <-> ENC Status compact/Status/Set counter done
//     PlcTask Inputs/GVL_iXlinker.EtherCAT_Master_EPPxxxx.Beckhoff_EPP5xxx.Beckhoff_EPP5xxxEK1122.A_0003_EPP5101_0002_0017.ENC_Status_compact.Status/Counter_underflow <-> ENC Status compact/Status/Counter underflow
//     PlcTask Inputs/GVL_iXlinker.EtherCAT_Master_EPPxxxx.Beckhoff_EPP5xxx.Beckhoff_EPP5xxxEK1122.A_0003_EPP5101_0002_0017.ENC_Status_compact.Status/Counter_overflow <-> ENC Status compact/Status/Counter overflow
//     PlcTask Inputs/GVL_iXlinker.EtherCAT_Master_EPPxxxx.Beckhoff_EPP5xxx.Beckhoff_EPP5xxxEK1122.A_0003_EPP5101_0002_0017.ENC_Status_compact.Status/Open_circuit <-> ENC Status compact/Status/Open circuit
//     PlcTask Inputs/GVL_iXlinker.EtherCAT_Master_EPPxxxx.Beckhoff_EPP5xxx.Beckhoff_EPP5xxxEK1122.A_0003_EPP5101_0002_0017.ENC_Status_compact.Status/Extrapolation_stall <-> ENC Status compact/Status/Extrapolation stall
//     PlcTask Inputs/GVL_iXlinker.EtherCAT_Master_EPPxxxx.Beckhoff_EPP5xxx.Beckhoff_EPP5xxxEK1122.A_0003_EPP5101_0002_0017.ENC_Status_compact.Status/Status_of_input_A <-> ENC Status compact/Status/Status of input A
//     PlcTask Inputs/GVL_iXlinker.EtherCAT_Master_EPPxxxx.Beckhoff_EPP5xxx.Beckhoff_EPP5xxxEK1122.A_0003_EPP5101_0002_0017.ENC_Status_compact.Status/Status_of_input_B <-> ENC Status compact/Status/Status of input B
//     PlcTask Inputs/GVL_iXlinker.EtherCAT_Master_EPPxxxx.Beckhoff_EPP5xxx.Beckhoff_EPP5xxxEK1122.A_0003_EPP5101_0002_0017.ENC_Status_compact.Status/Status_of_input_C <-> ENC Status compact/Status/Status of input C
//     PlcTask Inputs/GVL_iXlinker.EtherCAT_Master_EPPxxxx.Beckhoff_EPP5xxx.Beckhoff_EPP5xxxEK1122.A_0003_EPP5101_0002_0017.ENC_Status_compact.Status/Sync_error <-> ENC Status compact/Status/Sync error
//     PlcTask Inputs/GVL_iXlinker.EtherCAT_Master_EPPxxxx.Beckhoff_EPP5xxx.Beckhoff_EPP5xxxEK1122.A_0003_EPP5101_0002_0017.ENC_Status_compact.Status/TxPDO_State <-> ENC Status compact/Status/TxPDO State
//     PlcTask Inputs/GVL_iXlinker.EtherCAT_Master_EPPxxxx.Beckhoff_EPP5xxx.Beckhoff_EPP5xxxEK1122.A_0003_EPP5101_0002_0017.ENC_Status_compact.Status/TxPDO_Toggle <-> ENC Status compact/Status/TxPDO Toggle
//     PlcTask Inputs/GVL_iXlinker.EtherCAT_Master_EPPxxxx.Beckhoff_EPP5xxx.Beckhoff_EPP5xxxEK1122.A_0003_EPP5101_0002_0017.ENC_Status_compact.Counter_value <-> ENC Status compact/Counter value
//     PlcTask Inputs/GVL_iXlinker.EtherCAT_Master_EPPxxxx.Beckhoff_EPP5xxx.Beckhoff_EPP5xxxEK1122.A_0003_EPP5101_0002_0017.ENC_Status_compact.Latch_value <-> ENC Status compact/Latch value
//     PlcTask Outputs/GVL_iXlinker.EtherCAT_Master_EPPxxxx.Beckhoff_EPP5xxx.Beckhoff_EPP5xxxEK1122.A_0003_EPP5101_0002_0017.ENC_Control_compact.Control/Enable_latch_C <-> ENC Control compact/Control/Enable latch C
//     PlcTask Outputs/GVL_iXlinker.EtherCAT_Master_EPPxxxx.Beckhoff_EPP5xxx.Beckhoff_EPP5xxxEK1122.A_0003_EPP5101_0002_0017.ENC_Control_compact.Control/Set_counter <-> ENC Control compact/Control/Set counter
//     PlcTask Outputs/GVL_iXlinker.EtherCAT_Master_EPPxxxx.Beckhoff_EPP5xxx.Beckhoff_EPP5xxxEK1122.A_0003_EPP5101_0002_0017.ENC_Control_compact.Set_counter_value <-> ENC Control compact/Set counter value
//     PlcTask Inputs/GVL_iXlinker.EtherCAT_Master_EPPxxxx.Beckhoff_EPP5xxx.Beckhoff_EPP5xxxEK1122.A_0003_EPP5101_0002_0017.WcState.WcState <-> WcState/WcState
//     PlcTask Inputs/GVL_iXlinker.EtherCAT_Master_EPPxxxx.Beckhoff_EPP5xxx.Beckhoff_EPP5xxxEK1122.A_0003_EPP5101_0002_0017.WcState.InputToggle <-> WcState/InputToggle
//     PlcTask Inputs/GVL_iXlinker.EtherCAT_Master_EPPxxxx.Beckhoff_EPP5xxx.Beckhoff_EPP5xxxEK1122.A_0003_EPP5101_0002_0017.InfoData.AdsAddr <-> InfoData/AdsAddr
//     PlcTask Inputs/GVL_iXlinker.EtherCAT_Master_EPPxxxx.Beckhoff_EPP5xxx.Beckhoff_EPP5xxxEK1122.A_0003_EPP5101_0002_0017.InfoData.State <-> InfoData/State
//   PLC/PLC Instance <-> EtherCAT Master EPPxxxx/Beckhoff EPP5xxx/Beckhoff EPP5xxxEK1122/A_0004(EPP5101-0011-0016)
//     PlcTask Inputs/GVL_iXlinker.EtherCAT_Master_EPPxxxx.Beckhoff_EPP5xxx.Beckhoff_EPP5xxxEK1122.A_0004_EPP5101_0011_0016.ENC_Status_compact.Status/Latch_C_valid <-> ENC Status compact/Status/Latch C valid
//     PlcTask Inputs/GVL_iXlinker.EtherCAT_Master_EPPxxxx.Beckhoff_EPP5xxx.Beckhoff_EPP5xxxEK1122.A_0004_EPP5101_0011_0016.ENC_Status_compact.Status/Latch_extern_valid <-> ENC Status compact/Status/Latch extern valid
//     PlcTask Inputs/GVL_iXlinker.EtherCAT_Master_EPPxxxx.Beckhoff_EPP5xxx.Beckhoff_EPP5xxxEK1122.A_0004_EPP5101_0011_0016.ENC_Status_compact.Status/Set_counter_done <-> ENC Status compact/Status/Set counter done
//     PlcTask Inputs/GVL_iXlinker.EtherCAT_Master_EPPxxxx.Beckhoff_EPP5xxx.Beckhoff_EPP5xxxEK1122.A_0004_EPP5101_0011_0016.ENC_Status_compact.Status/Counter_underflow <-> ENC Status compact/Status/Counter underflow
//     PlcTask Inputs/GVL_iXlinker.EtherCAT_Master_EPPxxxx.Beckhoff_EPP5xxx.Beckhoff_EPP5xxxEK1122.A_0004_EPP5101_0011_0016.ENC_Status_compact.Status/Counter_overflow <-> ENC Status compact/Status/Counter overflow
//     PlcTask Inputs/GVL_iXlinker.EtherCAT_Master_EPPxxxx.Beckhoff_EPP5xxx.Beckhoff_EPP5xxxEK1122.A_0004_EPP5101_0011_0016.ENC_Status_compact.Status/Status_of_input_status <-> ENC Status compact/Status/Status of input status
//     PlcTask Inputs/GVL_iXlinker.EtherCAT_Master_EPPxxxx.Beckhoff_EPP5xxx.Beckhoff_EPP5xxxEK1122.A_0004_EPP5101_0011_0016.ENC_Status_compact.Status/Open_circuit <-> ENC Status compact/Status/Open circuit
//     PlcTask Inputs/GVL_iXlinker.EtherCAT_Master_EPPxxxx.Beckhoff_EPP5xxx.Beckhoff_EPP5xxxEK1122.A_0004_EPP5101_0011_0016.ENC_Status_compact.Status/Extrapolation_stall <-> ENC Status compact/Status/Extrapolation stall
//     PlcTask Inputs/GVL_iXlinker.EtherCAT_Master_EPPxxxx.Beckhoff_EPP5xxx.Beckhoff_EPP5xxxEK1122.A_0004_EPP5101_0011_0016.ENC_Status_compact.Status/Status_of_input_A <-> ENC Status compact/Status/Status of input A
//     PlcTask Inputs/GVL_iXlinker.EtherCAT_Master_EPPxxxx.Beckhoff_EPP5xxx.Beckhoff_EPP5xxxEK1122.A_0004_EPP5101_0011_0016.ENC_Status_compact.Status/Status_of_input_B <-> ENC Status compact/Status/Status of input B
//     PlcTask Inputs/GVL_iXlinker.EtherCAT_Master_EPPxxxx.Beckhoff_EPP5xxx.Beckhoff_EPP5xxxEK1122.A_0004_EPP5101_0011_0016.ENC_Status_compact.Status/Status_of_input_C <-> ENC Status compact/Status/Status of input C
//     PlcTask Inputs/GVL_iXlinker.EtherCAT_Master_EPPxxxx.Beckhoff_EPP5xxx.Beckhoff_EPP5xxxEK1122.A_0004_EPP5101_0011_0016.ENC_Status_compact.Status/Status_of_input_gate <-> ENC Status compact/Status/Status of input gate
//     PlcTask Inputs/GVL_iXlinker.EtherCAT_Master_EPPxxxx.Beckhoff_EPP5xxx.Beckhoff_EPP5xxxEK1122.A_0004_EPP5101_0011_0016.ENC_Status_compact.Status/Status_of_extern_latch <-> ENC Status compact/Status/Status of extern latch
//     PlcTask Inputs/GVL_iXlinker.EtherCAT_Master_EPPxxxx.Beckhoff_EPP5xxx.Beckhoff_EPP5xxxEK1122.A_0004_EPP5101_0011_0016.ENC_Status_compact.Status/Sync_error <-> ENC Status compact/Status/Sync error
//     PlcTask Inputs/GVL_iXlinker.EtherCAT_Master_EPPxxxx.Beckhoff_EPP5xxx.Beckhoff_EPP5xxxEK1122.A_0004_EPP5101_0011_0016.ENC_Status_compact.Status/TxPDO_State <-> ENC Status compact/Status/TxPDO State
//     PlcTask Inputs/GVL_iXlinker.EtherCAT_Master_EPPxxxx.Beckhoff_EPP5xxx.Beckhoff_EPP5xxxEK1122.A_0004_EPP5101_0011_0016.ENC_Status_compact.Status/TxPDO_Toggle <-> ENC Status compact/Status/TxPDO Toggle
//     PlcTask Inputs/GVL_iXlinker.EtherCAT_Master_EPPxxxx.Beckhoff_EPP5xxx.Beckhoff_EPP5xxxEK1122.A_0004_EPP5101_0011_0016.ENC_Status_compact.Counter_value <-> ENC Status compact/Counter value
//     PlcTask Inputs/GVL_iXlinker.EtherCAT_Master_EPPxxxx.Beckhoff_EPP5xxx.Beckhoff_EPP5xxxEK1122.A_0004_EPP5101_0011_0016.ENC_Status_compact.Latch_value <-> ENC Status compact/Latch value
//     PlcTask Outputs/GVL_iXlinker.EtherCAT_Master_EPPxxxx.Beckhoff_EPP5xxx.Beckhoff_EPP5xxxEK1122.A_0004_EPP5101_0011_0016.ENC_Control_compact.Control/Enable_latch_C <-> ENC Control compact/Control/Enable latch C
//     PlcTask Outputs/GVL_iXlinker.EtherCAT_Master_EPPxxxx.Beckhoff_EPP5xxx.Beckhoff_EPP5xxxEK1122.A_0004_EPP5101_0011_0016.ENC_Control_compact.Control/Enable_latch_extern_on_positive_edge <-> ENC Control compact/Control/Enable latch extern on positive edge
//     PlcTask Outputs/GVL_iXlinker.EtherCAT_Master_EPPxxxx.Beckhoff_EPP5xxx.Beckhoff_EPP5xxxEK1122.A_0004_EPP5101_0011_0016.ENC_Control_compact.Control/Set_counter <-> ENC Control compact/Control/Set counter
//     PlcTask Outputs/GVL_iXlinker.EtherCAT_Master_EPPxxxx.Beckhoff_EPP5xxx.Beckhoff_EPP5xxxEK1122.A_0004_EPP5101_0011_0016.ENC_Control_compact.Control/Enable_latch_extern_on_negative_edge <-> ENC Control compact/Control/Enable latch extern on negative edge
//     PlcTask Outputs/GVL_iXlinker.EtherCAT_Master_EPPxxxx.Beckhoff_EPP5xxx.Beckhoff_EPP5xxxEK1122.A_0004_EPP5101_0011_0016.ENC_Control_compact.Set_counter_value <-> ENC Control compact/Set counter value
//     PlcTask Inputs/GVL_iXlinker.EtherCAT_Master_EPPxxxx.Beckhoff_EPP5xxx.Beckhoff_EPP5xxxEK1122.A_0004_EPP5101_0011_0016.WcState.WcState <-> WcState/WcState
//     PlcTask Inputs/GVL_iXlinker.EtherCAT_Master_EPPxxxx.Beckhoff_EPP5xxx.Beckhoff_EPP5xxxEK1122.A_0004_EPP5101_0011_0016.WcState.InputToggle <-> WcState/InputToggle
//     PlcTask Inputs/GVL_iXlinker.EtherCAT_Master_EPPxxxx.Beckhoff_EPP5xxx.Beckhoff_EPP5xxxEK1122.A_0004_EPP5101_0011_0016.InfoData.AdsAddr <-> InfoData/AdsAddr
//     PlcTask Inputs/GVL_iXlinker.EtherCAT_Master_EPPxxxx.Beckhoff_EPP5xxx.Beckhoff_EPP5xxxEK1122.A_0004_EPP5101_0011_0016.InfoData.State <-> InfoData/State
//   PLC/PLC Instance <-> EtherCAT Master EPPxxxx/Beckhoff EPP5xxx/Beckhoff EPP5xxxEK1122/A_0005(EPP5101-0011-0017)
//     PlcTask Inputs/GVL_iXlinker.EtherCAT_Master_EPPxxxx.Beckhoff_EPP5xxx.Beckhoff_EPP5xxxEK1122.A_0005_EPP5101_0011_0017.ENC_Status_compact.Status/Latch_C_valid <-> ENC Status compact/Status/Latch C valid
//     PlcTask Inputs/GVL_iXlinker.EtherCAT_Master_EPPxxxx.Beckhoff_EPP5xxx.Beckhoff_EPP5xxxEK1122.A_0005_EPP5101_0011_0017.ENC_Status_compact.Status/Latch_extern_valid <-> ENC Status compact/Status/Latch extern valid
//     PlcTask Inputs/GVL_iXlinker.EtherCAT_Master_EPPxxxx.Beckhoff_EPP5xxx.Beckhoff_EPP5xxxEK1122.A_0005_EPP5101_0011_0017.ENC_Status_compact.Status/Set_counter_done <-> ENC Status compact/Status/Set counter done
//     PlcTask Inputs/GVL_iXlinker.EtherCAT_Master_EPPxxxx.Beckhoff_EPP5xxx.Beckhoff_EPP5xxxEK1122.A_0005_EPP5101_0011_0017.ENC_Status_compact.Status/Counter_underflow <-> ENC Status compact/Status/Counter underflow
//     PlcTask Inputs/GVL_iXlinker.EtherCAT_Master_EPPxxxx.Beckhoff_EPP5xxx.Beckhoff_EPP5xxxEK1122.A_0005_EPP5101_0011_0017.ENC_Status_compact.Status/Counter_overflow <-> ENC Status compact/Status/Counter overflow
//     PlcTask Inputs/GVL_iXlinker.EtherCAT_Master_EPPxxxx.Beckhoff_EPP5xxx.Beckhoff_EPP5xxxEK1122.A_0005_EPP5101_0011_0017.ENC_Status_compact.Status/Status_of_input_status <-> ENC Status compact/Status/Status of input status
//     PlcTask Inputs/GVL_iXlinker.EtherCAT_Master_EPPxxxx.Beckhoff_EPP5xxx.Beckhoff_EPP5xxxEK1122.A_0005_EPP5101_0011_0017.ENC_Status_compact.Status/Open_circuit <-> ENC Status compact/Status/Open circuit
//     PlcTask Inputs/GVL_iXlinker.EtherCAT_Master_EPPxxxx.Beckhoff_EPP5xxx.Beckhoff_EPP5xxxEK1122.A_0005_EPP5101_0011_0017.ENC_Status_compact.Status/Extrapolation_stall <-> ENC Status compact/Status/Extrapolation stall
//     PlcTask Inputs/GVL_iXlinker.EtherCAT_Master_EPPxxxx.Beckhoff_EPP5xxx.Beckhoff_EPP5xxxEK1122.A_0005_EPP5101_0011_0017.ENC_Status_compact.Status/Status_of_input_A <-> ENC Status compact/Status/Status of input A
//     PlcTask Inputs/GVL_iXlinker.EtherCAT_Master_EPPxxxx.Beckhoff_EPP5xxx.Beckhoff_EPP5xxxEK1122.A_0005_EPP5101_0011_0017.ENC_Status_compact.Status/Status_of_input_B <-> ENC Status compact/Status/Status of input B
//     PlcTask Inputs/GVL_iXlinker.EtherCAT_Master_EPPxxxx.Beckhoff_EPP5xxx.Beckhoff_EPP5xxxEK1122.A_0005_EPP5101_0011_0017.ENC_Status_compact.Status/Status_of_input_C <-> ENC Status compact/Status/Status of input C
//     PlcTask Inputs/GVL_iXlinker.EtherCAT_Master_EPPxxxx.Beckhoff_EPP5xxx.Beckhoff_EPP5xxxEK1122.A_0005_EPP5101_0011_0017.ENC_Status_compact.Status/Status_of_input_gate <-> ENC Status compact/Status/Status of input gate
//     PlcTask Inputs/GVL_iXlinker.EtherCAT_Master_EPPxxxx.Beckhoff_EPP5xxx.Beckhoff_EPP5xxxEK1122.A_0005_EPP5101_0011_0017.ENC_Status_compact.Status/Status_of_extern_latch <-> ENC Status compact/Status/Status of extern latch
//     PlcTask Inputs/GVL_iXlinker.EtherCAT_Master_EPPxxxx.Beckhoff_EPP5xxx.Beckhoff_EPP5xxxEK1122.A_0005_EPP5101_0011_0017.ENC_Status_compact.Status/Sync_error <-> ENC Status compact/Status/Sync error
//     PlcTask Inputs/GVL_iXlinker.EtherCAT_Master_EPPxxxx.Beckhoff_EPP5xxx.Beckhoff_EPP5xxxEK1122.A_0005_EPP5101_0011_0017.ENC_Status_compact.Status/TxPDO_State <-> ENC Status compact/Status/TxPDO State
//     PlcTask Inputs/GVL_iXlinker.EtherCAT_Master_EPPxxxx.Beckhoff_EPP5xxx.Beckhoff_EPP5xxxEK1122.A_0005_EPP5101_0011_0017.ENC_Status_compact.Status/TxPDO_Toggle <-> ENC Status compact/Status/TxPDO Toggle
//     PlcTask Inputs/GVL_iXlinker.EtherCAT_Master_EPPxxxx.Beckhoff_EPP5xxx.Beckhoff_EPP5xxxEK1122.A_0005_EPP5101_0011_0017.ENC_Status_compact.Counter_value <-> ENC Status compact/Counter value
//     PlcTask Inputs/GVL_iXlinker.EtherCAT_Master_EPPxxxx.Beckhoff_EPP5xxx.Beckhoff_EPP5xxxEK1122.A_0005_EPP5101_0011_0017.ENC_Status_compact.Latch_value <-> ENC Status compact/Latch value
//     PlcTask Outputs/GVL_iXlinker.EtherCAT_Master_EPPxxxx.Beckhoff_EPP5xxx.Beckhoff_EPP5xxxEK1122.A_0005_EPP5101_0011_0017.ENC_Control_compact.Control/Enable_latch_C <-> ENC Control compact/Control/Enable latch C
//     PlcTask Outputs/GVL_iXlinker.EtherCAT_Master_EPPxxxx.Beckhoff_EPP5xxx.Beckhoff_EPP5xxxEK1122.A_0005_EPP5101_0011_0017.ENC_Control_compact.Control/Enable_latch_extern_on_positive_edge <-> ENC Control compact/Control/Enable latch extern on positive edge
//     PlcTask Outputs/GVL_iXlinker.EtherCAT_Master_EPPxxxx.Beckhoff_EPP5xxx.Beckhoff_EPP5xxxEK1122.A_0005_EPP5101_0011_0017.ENC_Control_compact.Control/Set_counter <-> ENC Control compact/Control/Set counter
//     PlcTask Outputs/GVL_iXlinker.EtherCAT_Master_EPPxxxx.Beckhoff_EPP5xxx.Beckhoff_EPP5xxxEK1122.A_0005_EPP5101_0011_0017.ENC_Control_compact.Control/Enable_latch_extern_on_negative_edge <-> ENC Control compact/Control/Enable latch extern on negative edge
//     PlcTask Outputs/GVL_iXlinker.EtherCAT_Master_EPPxxxx.Beckhoff_EPP5xxx.Beckhoff_EPP5xxxEK1122.A_0005_EPP5101_0011_0017.ENC_Control_compact.Set_counter_value <-> ENC Control compact/Set counter value
//     PlcTask Inputs/GVL_iXlinker.EtherCAT_Master_EPPxxxx.Beckhoff_EPP5xxx.Beckhoff_EPP5xxxEK1122.A_0005_EPP5101_0011_0017.WcState.WcState <-> WcState/WcState
//     PlcTask Inputs/GVL_iXlinker.EtherCAT_Master_EPPxxxx.Beckhoff_EPP5xxx.Beckhoff_EPP5xxxEK1122.A_0005_EPP5101_0011_0017.WcState.InputToggle <-> WcState/InputToggle
//     PlcTask Inputs/GVL_iXlinker.EtherCAT_Master_EPPxxxx.Beckhoff_EPP5xxx.Beckhoff_EPP5xxxEK1122.A_0005_EPP5101_0011_0017.InfoData.AdsAddr <-> InfoData/AdsAddr
//     PlcTask Inputs/GVL_iXlinker.EtherCAT_Master_EPPxxxx.Beckhoff_EPP5xxx.Beckhoff_EPP5xxxEK1122.A_0005_EPP5101_0011_0017.InfoData.State <-> InfoData/State
//   PLC/PLC Instance <-> EtherCAT Master EPPxxxx/Beckhoff EPP5xxx/Beckhoff EPP5xxxEK1122/A_0006(EPP5101-1002-0016)
//     PlcTask Inputs/GVL_iXlinker.EtherCAT_Master_EPPxxxx.Beckhoff_EPP5xxx.Beckhoff_EPP5xxxEK1122.A_0006_EPP5101_1002_0016.ENC_Status_compact.Status/Latch_C_valid <-> ENC Status compact/Status/Latch C valid
//     PlcTask Inputs/GVL_iXlinker.EtherCAT_Master_EPPxxxx.Beckhoff_EPP5xxx.Beckhoff_EPP5xxxEK1122.A_0006_EPP5101_1002_0016.ENC_Status_compact.Status/Set_counter_done <-> ENC Status compact/Status/Set counter done
//     PlcTask Inputs/GVL_iXlinker.EtherCAT_Master_EPPxxxx.Beckhoff_EPP5xxx.Beckhoff_EPP5xxxEK1122.A_0006_EPP5101_1002_0016.ENC_Status_compact.Status/Counter_underflow <-> ENC Status compact/Status/Counter underflow
//     PlcTask Inputs/GVL_iXlinker.EtherCAT_Master_EPPxxxx.Beckhoff_EPP5xxx.Beckhoff_EPP5xxxEK1122.A_0006_EPP5101_1002_0016.ENC_Status_compact.Status/Counter_overflow <-> ENC Status compact/Status/Counter overflow
//     PlcTask Inputs/GVL_iXlinker.EtherCAT_Master_EPPxxxx.Beckhoff_EPP5xxx.Beckhoff_EPP5xxxEK1122.A_0006_EPP5101_1002_0016.ENC_Status_compact.Status/Open_circuit <-> ENC Status compact/Status/Open circuit
//     PlcTask Inputs/GVL_iXlinker.EtherCAT_Master_EPPxxxx.Beckhoff_EPP5xxx.Beckhoff_EPP5xxxEK1122.A_0006_EPP5101_1002_0016.ENC_Status_compact.Status/Extrapolation_stall <-> ENC Status compact/Status/Extrapolation stall
//     PlcTask Inputs/GVL_iXlinker.EtherCAT_Master_EPPxxxx.Beckhoff_EPP5xxx.Beckhoff_EPP5xxxEK1122.A_0006_EPP5101_1002_0016.ENC_Status_compact.Status/Status_of_input_A <-> ENC Status compact/Status/Status of input A
//     PlcTask Inputs/GVL_iXlinker.EtherCAT_Master_EPPxxxx.Beckhoff_EPP5xxx.Beckhoff_EPP5xxxEK1122.A_0006_EPP5101_1002_0016.ENC_Status_compact.Status/Status_of_input_B <-> ENC Status compact/Status/Status of input B
//     PlcTask Inputs/GVL_iXlinker.EtherCAT_Master_EPPxxxx.Beckhoff_EPP5xxx.Beckhoff_EPP5xxxEK1122.A_0006_EPP5101_1002_0016.ENC_Status_compact.Status/Status_of_input_C <-> ENC Status compact/Status/Status of input C
//     PlcTask Inputs/GVL_iXlinker.EtherCAT_Master_EPPxxxx.Beckhoff_EPP5xxx.Beckhoff_EPP5xxxEK1122.A_0006_EPP5101_1002_0016.ENC_Status_compact.Status/Sync_error <-> ENC Status compact/Status/Sync error
//     PlcTask Inputs/GVL_iXlinker.EtherCAT_Master_EPPxxxx.Beckhoff_EPP5xxx.Beckhoff_EPP5xxxEK1122.A_0006_EPP5101_1002_0016.ENC_Status_compact.Status/TxPDO_State <-> ENC Status compact/Status/TxPDO State
//     PlcTask Inputs/GVL_iXlinker.EtherCAT_Master_EPPxxxx.Beckhoff_EPP5xxx.Beckhoff_EPP5xxxEK1122.A_0006_EPP5101_1002_0016.ENC_Status_compact.Status/TxPDO_Toggle <-> ENC Status compact/Status/TxPDO Toggle
//     PlcTask Inputs/GVL_iXlinker.EtherCAT_Master_EPPxxxx.Beckhoff_EPP5xxx.Beckhoff_EPP5xxxEK1122.A_0006_EPP5101_1002_0016.ENC_Status_compact.Counter_value <-> ENC Status compact/Counter value
//     PlcTask Inputs/GVL_iXlinker.EtherCAT_Master_EPPxxxx.Beckhoff_EPP5xxx.Beckhoff_EPP5xxxEK1122.A_0006_EPP5101_1002_0016.ENC_Status_compact.Latch_value <-> ENC Status compact/Latch value
//     PlcTask Outputs/GVL_iXlinker.EtherCAT_Master_EPPxxxx.Beckhoff_EPP5xxx.Beckhoff_EPP5xxxEK1122.A_0006_EPP5101_1002_0016.ENC_Control_compact.Control/Enable_latch_C <-> ENC Control compact/Control/Enable latch C
//     PlcTask Outputs/GVL_iXlinker.EtherCAT_Master_EPPxxxx.Beckhoff_EPP5xxx.Beckhoff_EPP5xxxEK1122.A_0006_EPP5101_1002_0016.ENC_Control_compact.Control/Set_counter <-> ENC Control compact/Control/Set counter
//     PlcTask Outputs/GVL_iXlinker.EtherCAT_Master_EPPxxxx.Beckhoff_EPP5xxx.Beckhoff_EPP5xxxEK1122.A_0006_EPP5101_1002_0016.ENC_Control_compact.Set_counter_value <-> ENC Control compact/Set counter value
//     PlcTask Inputs/GVL_iXlinker.EtherCAT_Master_EPPxxxx.Beckhoff_EPP5xxx.Beckhoff_EPP5xxxEK1122.A_0006_EPP5101_1002_0016.WcState.WcState <-> WcState/WcState
//     PlcTask Inputs/GVL_iXlinker.EtherCAT_Master_EPPxxxx.Beckhoff_EPP5xxx.Beckhoff_EPP5xxxEK1122.A_0006_EPP5101_1002_0016.WcState.InputToggle <-> WcState/InputToggle
//     PlcTask Inputs/GVL_iXlinker.EtherCAT_Master_EPPxxxx.Beckhoff_EPP5xxx.Beckhoff_EPP5xxxEK1122.A_0006_EPP5101_1002_0016.InfoData.AdsAddr <-> InfoData/AdsAddr
//     PlcTask Inputs/GVL_iXlinker.EtherCAT_Master_EPPxxxx.Beckhoff_EPP5xxx.Beckhoff_EPP5xxxEK1122.A_0006_EPP5101_1002_0016.InfoData.State <-> InfoData/State
//   PLC/PLC Instance <-> EtherCAT Master EPPxxxx/Beckhoff EPP5xxx/Beckhoff EPP5xxxEK1122/A_0007(EPP5101-1002-0017)
//     PlcTask Inputs/GVL_iXlinker.EtherCAT_Master_EPPxxxx.Beckhoff_EPP5xxx.Beckhoff_EPP5xxxEK1122.A_0007_EPP5101_1002_0017.ENC_Status_compact.Status/Latch_C_valid <-> ENC Status compact/Status/Latch C valid
//     PlcTask Inputs/GVL_iXlinker.EtherCAT_Master_EPPxxxx.Beckhoff_EPP5xxx.Beckhoff_EPP5xxxEK1122.A_0007_EPP5101_1002_0017.ENC_Status_compact.Status/Set_counter_done <-> ENC Status compact/Status/Set counter done
//     PlcTask Inputs/GVL_iXlinker.EtherCAT_Master_EPPxxxx.Beckhoff_EPP5xxx.Beckhoff_EPP5xxxEK1122.A_0007_EPP5101_1002_0017.ENC_Status_compact.Status/Counter_underflow <-> ENC Status compact/Status/Counter underflow
//     PlcTask Inputs/GVL_iXlinker.EtherCAT_Master_EPPxxxx.Beckhoff_EPP5xxx.Beckhoff_EPP5xxxEK1122.A_0007_EPP5101_1002_0017.ENC_Status_compact.Status/Counter_overflow <-> ENC Status compact/Status/Counter overflow
//     PlcTask Inputs/GVL_iXlinker.EtherCAT_Master_EPPxxxx.Beckhoff_EPP5xxx.Beckhoff_EPP5xxxEK1122.A_0007_EPP5101_1002_0017.ENC_Status_compact.Status/Open_circuit <-> ENC Status compact/Status/Open circuit
//     PlcTask Inputs/GVL_iXlinker.EtherCAT_Master_EPPxxxx.Beckhoff_EPP5xxx.Beckhoff_EPP5xxxEK1122.A_0007_EPP5101_1002_0017.ENC_Status_compact.Status/Extrapolation_stall <-> ENC Status compact/Status/Extrapolation stall
//     PlcTask Inputs/GVL_iXlinker.EtherCAT_Master_EPPxxxx.Beckhoff_EPP5xxx.Beckhoff_EPP5xxxEK1122.A_0007_EPP5101_1002_0017.ENC_Status_compact.Status/Status_of_input_A <-> ENC Status compact/Status/Status of input A
//     PlcTask Inputs/GVL_iXlinker.EtherCAT_Master_EPPxxxx.Beckhoff_EPP5xxx.Beckhoff_EPP5xxxEK1122.A_0007_EPP5101_1002_0017.ENC_Status_compact.Status/Status_of_input_B <-> ENC Status compact/Status/Status of input B
//     PlcTask Inputs/GVL_iXlinker.EtherCAT_Master_EPPxxxx.Beckhoff_EPP5xxx.Beckhoff_EPP5xxxEK1122.A_0007_EPP5101_1002_0017.ENC_Status_compact.Status/Status_of_input_C <-> ENC Status compact/Status/Status of input C
//     PlcTask Inputs/GVL_iXlinker.EtherCAT_Master_EPPxxxx.Beckhoff_EPP5xxx.Beckhoff_EPP5xxxEK1122.A_0007_EPP5101_1002_0017.ENC_Status_compact.Status/Sync_error <-> ENC Status compact/Status/Sync error
//     PlcTask Inputs/GVL_iXlinker.EtherCAT_Master_EPPxxxx.Beckhoff_EPP5xxx.Beckhoff_EPP5xxxEK1122.A_0007_EPP5101_1002_0017.ENC_Status_compact.Status/TxPDO_State <-> ENC Status compact/Status/TxPDO State
//     PlcTask Inputs/GVL_iXlinker.EtherCAT_Master_EPPxxxx.Beckhoff_EPP5xxx.Beckhoff_EPP5xxxEK1122.A_0007_EPP5101_1002_0017.ENC_Status_compact.Status/TxPDO_Toggle <-> ENC Status compact/Status/TxPDO Toggle
//     PlcTask Inputs/GVL_iXlinker.EtherCAT_Master_EPPxxxx.Beckhoff_EPP5xxx.Beckhoff_EPP5xxxEK1122.A_0007_EPP5101_1002_0017.ENC_Status_compact.Counter_value <-> ENC Status compact/Counter value
//     PlcTask Inputs/GVL_iXlinker.EtherCAT_Master_EPPxxxx.Beckhoff_EPP5xxx.Beckhoff_EPP5xxxEK1122.A_0007_EPP5101_1002_0017.ENC_Status_compact.Latch_value <-> ENC Status compact/Latch value
//     PlcTask Outputs/GVL_iXlinker.EtherCAT_Master_EPPxxxx.Beckhoff_EPP5xxx.Beckhoff_EPP5xxxEK1122.A_0007_EPP5101_1002_0017.ENC_Control_compact.Control/Enable_latch_C <-> ENC Control compact/Control/Enable latch C
//     PlcTask Outputs/GVL_iXlinker.EtherCAT_Master_EPPxxxx.Beckhoff_EPP5xxx.Beckhoff_EPP5xxxEK1122.A_0007_EPP5101_1002_0017.ENC_Control_compact.Control/Set_counter <-> ENC Control compact/Control/Set counter
//     PlcTask Outputs/GVL_iXlinker.EtherCAT_Master_EPPxxxx.Beckhoff_EPP5xxx.Beckhoff_EPP5xxxEK1122.A_0007_EPP5101_1002_0017.ENC_Control_compact.Set_counter_value <-> ENC Control compact/Set counter value
//     PlcTask Inputs/GVL_iXlinker.EtherCAT_Master_EPPxxxx.Beckhoff_EPP5xxx.Beckhoff_EPP5xxxEK1122.A_0007_EPP5101_1002_0017.WcState.WcState <-> WcState/WcState
//     PlcTask Inputs/GVL_iXlinker.EtherCAT_Master_EPPxxxx.Beckhoff_EPP5xxx.Beckhoff_EPP5xxxEK1122.A_0007_EPP5101_1002_0017.WcState.InputToggle <-> WcState/InputToggle
//     PlcTask Inputs/GVL_iXlinker.EtherCAT_Master_EPPxxxx.Beckhoff_EPP5xxx.Beckhoff_EPP5xxxEK1122.A_0007_EPP5101_1002_0017.InfoData.AdsAddr <-> InfoData/AdsAddr
//     PlcTask Inputs/GVL_iXlinker.EtherCAT_Master_EPPxxxx.Beckhoff_EPP5xxx.Beckhoff_EPP5xxxEK1122.A_0007_EPP5101_1002_0017.InfoData.State <-> InfoData/State
//   PLC/PLC Instance <-> EtherCAT Master EPPxxxx/Beckhoff EPP5xxx/Beckhoff EPP5xxxEK1122/A_0008(EPP5151-0002-0016)
//     PlcTask Inputs/GVL_iXlinker.EtherCAT_Master_EPPxxxx.Beckhoff_EPP5xxx.Beckhoff_EPP5xxxEK1122.A_0008_EPP5151_0002_0016.ENC_Status_compact.Status/Latch_C_valid <-> ENC Status compact/Status/Latch C valid
//     PlcTask Inputs/GVL_iXlinker.EtherCAT_Master_EPPxxxx.Beckhoff_EPP5xxx.Beckhoff_EPP5xxxEK1122.A_0008_EPP5151_0002_0016.ENC_Status_compact.Status/Latch_extern_valid <-> ENC Status compact/Status/Latch extern valid
//     PlcTask Inputs/GVL_iXlinker.EtherCAT_Master_EPPxxxx.Beckhoff_EPP5xxx.Beckhoff_EPP5xxxEK1122.A_0008_EPP5151_0002_0016.ENC_Status_compact.Status/Set_counter_done <-> ENC Status compact/Status/Set counter done
//     PlcTask Inputs/GVL_iXlinker.EtherCAT_Master_EPPxxxx.Beckhoff_EPP5xxx.Beckhoff_EPP5xxxEK1122.A_0008_EPP5151_0002_0016.ENC_Status_compact.Status/Counter_underflow <-> ENC Status compact/Status/Counter underflow
//     PlcTask Inputs/GVL_iXlinker.EtherCAT_Master_EPPxxxx.Beckhoff_EPP5xxx.Beckhoff_EPP5xxxEK1122.A_0008_EPP5151_0002_0016.ENC_Status_compact.Status/Counter_overflow <-> ENC Status compact/Status/Counter overflow
//     PlcTask Inputs/GVL_iXlinker.EtherCAT_Master_EPPxxxx.Beckhoff_EPP5xxx.Beckhoff_EPP5xxxEK1122.A_0008_EPP5151_0002_0016.ENC_Status_compact.Status/Status_of_input_status <-> ENC Status compact/Status/Status of input status
//     PlcTask Inputs/GVL_iXlinker.EtherCAT_Master_EPPxxxx.Beckhoff_EPP5xxx.Beckhoff_EPP5xxxEK1122.A_0008_EPP5151_0002_0016.ENC_Status_compact.Status/Open_circuit <-> ENC Status compact/Status/Open circuit
//     PlcTask Inputs/GVL_iXlinker.EtherCAT_Master_EPPxxxx.Beckhoff_EPP5xxx.Beckhoff_EPP5xxxEK1122.A_0008_EPP5151_0002_0016.ENC_Status_compact.Status/Extrapolation_stall <-> ENC Status compact/Status/Extrapolation stall
//     PlcTask Inputs/GVL_iXlinker.EtherCAT_Master_EPPxxxx.Beckhoff_EPP5xxx.Beckhoff_EPP5xxxEK1122.A_0008_EPP5151_0002_0016.ENC_Status_compact.Status/Status_of_input_A <-> ENC Status compact/Status/Status of input A
//     PlcTask Inputs/GVL_iXlinker.EtherCAT_Master_EPPxxxx.Beckhoff_EPP5xxx.Beckhoff_EPP5xxxEK1122.A_0008_EPP5151_0002_0016.ENC_Status_compact.Status/Status_of_input_B <-> ENC Status compact/Status/Status of input B
//     PlcTask Inputs/GVL_iXlinker.EtherCAT_Master_EPPxxxx.Beckhoff_EPP5xxx.Beckhoff_EPP5xxxEK1122.A_0008_EPP5151_0002_0016.ENC_Status_compact.Status/Status_of_input_C <-> ENC Status compact/Status/Status of input C
//     PlcTask Inputs/GVL_iXlinker.EtherCAT_Master_EPPxxxx.Beckhoff_EPP5xxx.Beckhoff_EPP5xxxEK1122.A_0008_EPP5151_0002_0016.ENC_Status_compact.Status/Status_of_input_gate <-> ENC Status compact/Status/Status of input gate
//     PlcTask Inputs/GVL_iXlinker.EtherCAT_Master_EPPxxxx.Beckhoff_EPP5xxx.Beckhoff_EPP5xxxEK1122.A_0008_EPP5151_0002_0016.ENC_Status_compact.Status/Status_of_extern_latch <-> ENC Status compact/Status/Status of extern latch
//     PlcTask Inputs/GVL_iXlinker.EtherCAT_Master_EPPxxxx.Beckhoff_EPP5xxx.Beckhoff_EPP5xxxEK1122.A_0008_EPP5151_0002_0016.ENC_Status_compact.Status/Sync_error <-> ENC Status compact/Status/Sync error
//     PlcTask Inputs/GVL_iXlinker.EtherCAT_Master_EPPxxxx.Beckhoff_EPP5xxx.Beckhoff_EPP5xxxEK1122.A_0008_EPP5151_0002_0016.ENC_Status_compact.Status/TxPDO_State <-> ENC Status compact/Status/TxPDO State
//     PlcTask Inputs/GVL_iXlinker.EtherCAT_Master_EPPxxxx.Beckhoff_EPP5xxx.Beckhoff_EPP5xxxEK1122.A_0008_EPP5151_0002_0016.ENC_Status_compact.Status/TxPDO_Toggle <-> ENC Status compact/Status/TxPDO Toggle
//     PlcTask Inputs/GVL_iXlinker.EtherCAT_Master_EPPxxxx.Beckhoff_EPP5xxx.Beckhoff_EPP5xxxEK1122.A_0008_EPP5151_0002_0016.ENC_Status_compact.Counter_value <-> ENC Status compact/Counter value
//     PlcTask Inputs/GVL_iXlinker.EtherCAT_Master_EPPxxxx.Beckhoff_EPP5xxx.Beckhoff_EPP5xxxEK1122.A_0008_EPP5151_0002_0016.ENC_Status_compact.Latch_value <-> ENC Status compact/Latch value
//     PlcTask Outputs/GVL_iXlinker.EtherCAT_Master_EPPxxxx.Beckhoff_EPP5xxx.Beckhoff_EPP5xxxEK1122.A_0008_EPP5151_0002_0016.ENC_Control_compact.Control/Enable_latch_C <-> ENC Control compact/Control/Enable latch C
//     PlcTask Outputs/GVL_iXlinker.EtherCAT_Master_EPPxxxx.Beckhoff_EPP5xxx.Beckhoff_EPP5xxxEK1122.A_0008_EPP5151_0002_0016.ENC_Control_compact.Control/Enable_latch_extern_on_positive_edge <-> ENC Control compact/Control/Enable latch extern on positive edge
//     PlcTask Outputs/GVL_iXlinker.EtherCAT_Master_EPPxxxx.Beckhoff_EPP5xxx.Beckhoff_EPP5xxxEK1122.A_0008_EPP5151_0002_0016.ENC_Control_compact.Control/Set_counter <-> ENC Control compact/Control/Set counter
//     PlcTask Outputs/GVL_iXlinker.EtherCAT_Master_EPPxxxx.Beckhoff_EPP5xxx.Beckhoff_EPP5xxxEK1122.A_0008_EPP5151_0002_0016.ENC_Control_compact.Control/Enable_latch_extern_on_negative_edge <-> ENC Control compact/Control/Enable latch extern on negative edge
//     PlcTask Outputs/GVL_iXlinker.EtherCAT_Master_EPPxxxx.Beckhoff_EPP5xxx.Beckhoff_EPP5xxxEK1122.A_0008_EPP5151_0002_0016.ENC_Control_compact.Set_counter_value <-> ENC Control compact/Set counter value
//     PlcTask Inputs/GVL_iXlinker.EtherCAT_Master_EPPxxxx.Beckhoff_EPP5xxx.Beckhoff_EPP5xxxEK1122.A_0008_EPP5151_0002_0016.WcState.WcState <-> WcState/WcState
//     PlcTask Inputs/GVL_iXlinker.EtherCAT_Master_EPPxxxx.Beckhoff_EPP5xxx.Beckhoff_EPP5xxxEK1122.A_0008_EPP5151_0002_0016.WcState.InputToggle <-> WcState/InputToggle
//     PlcTask Inputs/GVL_iXlinker.EtherCAT_Master_EPPxxxx.Beckhoff_EPP5xxx.Beckhoff_EPP5xxxEK1122.A_0008_EPP5151_0002_0016.InfoData.AdsAddr <-> InfoData/AdsAddr
//     PlcTask Inputs/GVL_iXlinker.EtherCAT_Master_EPPxxxx.Beckhoff_EPP5xxx.Beckhoff_EPP5xxxEK1122.A_0008_EPP5151_0002_0016.InfoData.State <-> InfoData/State
//   PLC/PLC Instance <-> EtherCAT Master EPPxxxx/Beckhoff EPP5xxx/Beckhoff EPP5xxxEK1122/A_0009(EPP5151-0002-0017)
//     PlcTask Inputs/GVL_iXlinker.EtherCAT_Master_EPPxxxx.Beckhoff_EPP5xxx.Beckhoff_EPP5xxxEK1122.A_0009_EPP5151_0002_0017.ENC_Status_compact.Status/Latch_C_valid <-> ENC Status compact/Status/Latch C valid
//     PlcTask Inputs/GVL_iXlinker.EtherCAT_Master_EPPxxxx.Beckhoff_EPP5xxx.Beckhoff_EPP5xxxEK1122.A_0009_EPP5151_0002_0017.ENC_Status_compact.Status/Latch_extern_valid <-> ENC Status compact/Status/Latch extern valid
//     PlcTask Inputs/GVL_iXlinker.EtherCAT_Master_EPPxxxx.Beckhoff_EPP5xxx.Beckhoff_EPP5xxxEK1122.A_0009_EPP5151_0002_0017.ENC_Status_compact.Status/Set_counter_done <-> ENC Status compact/Status/Set counter done
//     PlcTask Inputs/GVL_iXlinker.EtherCAT_Master_EPPxxxx.Beckhoff_EPP5xxx.Beckhoff_EPP5xxxEK1122.A_0009_EPP5151_0002_0017.ENC_Status_compact.Status/Counter_underflow <-> ENC Status compact/Status/Counter underflow
//     PlcTask Inputs/GVL_iXlinker.EtherCAT_Master_EPPxxxx.Beckhoff_EPP5xxx.Beckhoff_EPP5xxxEK1122.A_0009_EPP5151_0002_0017.ENC_Status_compact.Status/Counter_overflow <-> ENC Status compact/Status/Counter overflow
//     PlcTask Inputs/GVL_iXlinker.EtherCAT_Master_EPPxxxx.Beckhoff_EPP5xxx.Beckhoff_EPP5xxxEK1122.A_0009_EPP5151_0002_0017.ENC_Status_compact.Status/Status_of_input_status <-> ENC Status compact/Status/Status of input status
//     PlcTask Inputs/GVL_iXlinker.EtherCAT_Master_EPPxxxx.Beckhoff_EPP5xxx.Beckhoff_EPP5xxxEK1122.A_0009_EPP5151_0002_0017.ENC_Status_compact.Status/Open_circuit <-> ENC Status compact/Status/Open circuit
//     PlcTask Inputs/GVL_iXlinker.EtherCAT_Master_EPPxxxx.Beckhoff_EPP5xxx.Beckhoff_EPP5xxxEK1122.A_0009_EPP5151_0002_0017.ENC_Status_compact.Status/Extrapolation_stall <-> ENC Status compact/Status/Extrapolation stall
//     PlcTask Inputs/GVL_iXlinker.EtherCAT_Master_EPPxxxx.Beckhoff_EPP5xxx.Beckhoff_EPP5xxxEK1122.A_0009_EPP5151_0002_0017.ENC_Status_compact.Status/Status_of_input_A <-> ENC Status compact/Status/Status of input A
//     PlcTask Inputs/GVL_iXlinker.EtherCAT_Master_EPPxxxx.Beckhoff_EPP5xxx.Beckhoff_EPP5xxxEK1122.A_0009_EPP5151_0002_0017.ENC_Status_compact.Status/Status_of_input_B <-> ENC Status compact/Status/Status of input B
//     PlcTask Inputs/GVL_iXlinker.EtherCAT_Master_EPPxxxx.Beckhoff_EPP5xxx.Beckhoff_EPP5xxxEK1122.A_0009_EPP5151_0002_0017.ENC_Status_compact.Status/Status_of_input_C <-> ENC Status compact/Status/Status of input C
//     PlcTask Inputs/GVL_iXlinker.EtherCAT_Master_EPPxxxx.Beckhoff_EPP5xxx.Beckhoff_EPP5xxxEK1122.A_0009_EPP5151_0002_0017.ENC_Status_compact.Status/Status_of_input_gate <-> ENC Status compact/Status/Status of input gate
//     PlcTask Inputs/GVL_iXlinker.EtherCAT_Master_EPPxxxx.Beckhoff_EPP5xxx.Beckhoff_EPP5xxxEK1122.A_0009_EPP5151_0002_0017.ENC_Status_compact.Status/Status_of_extern_latch <-> ENC Status compact/Status/Status of extern latch
//     PlcTask Inputs/GVL_iXlinker.EtherCAT_Master_EPPxxxx.Beckhoff_EPP5xxx.Beckhoff_EPP5xxxEK1122.A_0009_EPP5151_0002_0017.ENC_Status_compact.Status/Sync_error <-> ENC Status compact/Status/Sync error
//     PlcTask Inputs/GVL_iXlinker.EtherCAT_Master_EPPxxxx.Beckhoff_EPP5xxx.Beckhoff_EPP5xxxEK1122.A_0009_EPP5151_0002_0017.ENC_Status_compact.Status/TxPDO_State <-> ENC Status compact/Status/TxPDO State
//     PlcTask Inputs/GVL_iXlinker.EtherCAT_Master_EPPxxxx.Beckhoff_EPP5xxx.Beckhoff_EPP5xxxEK1122.A_0009_EPP5151_0002_0017.ENC_Status_compact.Status/TxPDO_Toggle <-> ENC Status compact/Status/TxPDO Toggle
//     PlcTask Inputs/GVL_iXlinker.EtherCAT_Master_EPPxxxx.Beckhoff_EPP5xxx.Beckhoff_EPP5xxxEK1122.A_0009_EPP5151_0002_0017.ENC_Status_compact.Counter_value <-> ENC Status compact/Counter value
//     PlcTask Inputs/GVL_iXlinker.EtherCAT_Master_EPPxxxx.Beckhoff_EPP5xxx.Beckhoff_EPP5xxxEK1122.A_0009_EPP5151_0002_0017.ENC_Status_compact.Latch_value <-> ENC Status compact/Latch value
//     PlcTask Outputs/GVL_iXlinker.EtherCAT_Master_EPPxxxx.Beckhoff_EPP5xxx.Beckhoff_EPP5xxxEK1122.A_0009_EPP5151_0002_0017.ENC_Control_compact.Control/Enable_latch_C <-> ENC Control compact/Control/Enable latch C
//     PlcTask Outputs/GVL_iXlinker.EtherCAT_Master_EPPxxxx.Beckhoff_EPP5xxx.Beckhoff_EPP5xxxEK1122.A_0009_EPP5151_0002_0017.ENC_Control_compact.Control/Enable_latch_extern_on_positive_edge <-> ENC Control compact/Control/Enable latch extern on positive edge
//     PlcTask Outputs/GVL_iXlinker.EtherCAT_Master_EPPxxxx.Beckhoff_EPP5xxx.Beckhoff_EPP5xxxEK1122.A_0009_EPP5151_0002_0017.ENC_Control_compact.Control/Set_counter <-> ENC Control compact/Control/Set counter
//     PlcTask Outputs/GVL_iXlinker.EtherCAT_Master_EPPxxxx.Beckhoff_EPP5xxx.Beckhoff_EPP5xxxEK1122.A_0009_EPP5151_0002_0017.ENC_Control_compact.Control/Enable_latch_extern_on_negative_edge <-> ENC Control compact/Control/Enable latch extern on negative edge
//     PlcTask Outputs/GVL_iXlinker.EtherCAT_Master_EPPxxxx.Beckhoff_EPP5xxx.Beckhoff_EPP5xxxEK1122.A_0009_EPP5151_0002_0017.ENC_Control_compact.Set_counter_value <-> ENC Control compact/Set counter value
//     PlcTask Inputs/GVL_iXlinker.EtherCAT_Master_EPPxxxx.Beckhoff_EPP5xxx.Beckhoff_EPP5xxxEK1122.A_0009_EPP5151_0002_0017.WcState.WcState <-> WcState/WcState
//     PlcTask Inputs/GVL_iXlinker.EtherCAT_Master_EPPxxxx.Beckhoff_EPP5xxx.Beckhoff_EPP5xxxEK1122.A_0009_EPP5151_0002_0017.WcState.InputToggle <-> WcState/InputToggle
//     PlcTask Inputs/GVL_iXlinker.EtherCAT_Master_EPPxxxx.Beckhoff_EPP5xxx.Beckhoff_EPP5xxxEK1122.A_0009_EPP5151_0002_0017.InfoData.AdsAddr <-> InfoData/AdsAddr
//     PlcTask Inputs/GVL_iXlinker.EtherCAT_Master_EPPxxxx.Beckhoff_EPP5xxx.Beckhoff_EPP5xxxEK1122.A_0009_EPP5151_0002_0017.InfoData.State <-> InfoData/State
//   PLC/PLC Instance <-> EtherCAT Master EPPxxxx/Beckhoff EPP6xxx
//     PlcTask Inputs/GVL_iXlinker.EtherCAT_Master_EPPxxxx.Beckhoff_EPP6xxx.InfoData.State <-> InfoData/State
//   PLC/PLC Instance <-> EtherCAT Master EPPxxxx/Beckhoff EPP6xxx/Beckhoff EPP6xxxEK1122
//     PlcTask Inputs/GVL_iXlinker.EtherCAT_Master_EPPxxxx.Beckhoff_EPP6xxx.Beckhoff_EPP6xxxEK1122.InfoData.State <-> InfoData/State
//   PLC/PLC Instance <-> EtherCAT Master EPPxxxx/Beckhoff EPP6xxx/Beckhoff EPP6xxxEK1122/Beckhoff EPP6xxxsub EK1100
//     PlcTask Inputs/GVL_iXlinker.EtherCAT_Master_EPPxxxx.Beckhoff_EPP6xxx.Beckhoff_EPP6xxxEK1122.Beckhoff_EPP6xxxsub_EK1100.InfoData.State <-> InfoData/State
//   PLC/PLC Instance <-> EtherCAT Master EPPxxxx/Beckhoff EPP6xxx/Beckhoff EPP6xxxEK1122/A_0001(EPP6001-0002-0016)
//     PlcTask Inputs/GVL_iXlinker.EtherCAT_Master_EPPxxxx.Beckhoff_EPP6xxx.Beckhoff_EPP6xxxEK1122.A_0001_EPP6001_0002_0016.COM_Inputs.Status <-> COM Inputs/Status
//     PlcTask Inputs/GVL_iXlinker.EtherCAT_Master_EPPxxxx.Beckhoff_EPP6xxx.Beckhoff_EPP6xxxEK1122.A_0001_EPP6001_0002_0016.COM_Inputs.Data_In[0] <-> COM Inputs/Data In 0
//     PlcTask Inputs/GVL_iXlinker.EtherCAT_Master_EPPxxxx.Beckhoff_EPP6xxx.Beckhoff_EPP6xxxEK1122.A_0001_EPP6001_0002_0016.COM_Inputs.Data_In[1] <-> COM Inputs/Data In 1
//     PlcTask Inputs/GVL_iXlinker.EtherCAT_Master_EPPxxxx.Beckhoff_EPP6xxx.Beckhoff_EPP6xxxEK1122.A_0001_EPP6001_0002_0016.COM_Inputs.Data_In[2] <-> COM Inputs/Data In 2
//     PlcTask Inputs/GVL_iXlinker.EtherCAT_Master_EPPxxxx.Beckhoff_EPP6xxx.Beckhoff_EPP6xxxEK1122.A_0001_EPP6001_0002_0016.COM_Inputs.Data_In[3] <-> COM Inputs/Data In 3
//     PlcTask Inputs/GVL_iXlinker.EtherCAT_Master_EPPxxxx.Beckhoff_EPP6xxx.Beckhoff_EPP6xxxEK1122.A_0001_EPP6001_0002_0016.COM_Inputs.Data_In[4] <-> COM Inputs/Data In 4
//     PlcTask Inputs/GVL_iXlinker.EtherCAT_Master_EPPxxxx.Beckhoff_EPP6xxx.Beckhoff_EPP6xxxEK1122.A_0001_EPP6001_0002_0016.COM_Inputs.Data_In[5] <-> COM Inputs/Data In 5
//     PlcTask Inputs/GVL_iXlinker.EtherCAT_Master_EPPxxxx.Beckhoff_EPP6xxx.Beckhoff_EPP6xxxEK1122.A_0001_EPP6001_0002_0016.COM_Inputs.Data_In[6] <-> COM Inputs/Data In 6
//     PlcTask Inputs/GVL_iXlinker.EtherCAT_Master_EPPxxxx.Beckhoff_EPP6xxx.Beckhoff_EPP6xxxEK1122.A_0001_EPP6001_0002_0016.COM_Inputs.Data_In[7] <-> COM Inputs/Data In 7
//     PlcTask Inputs/GVL_iXlinker.EtherCAT_Master_EPPxxxx.Beckhoff_EPP6xxx.Beckhoff_EPP6xxxEK1122.A_0001_EPP6001_0002_0016.COM_Inputs.Data_In[8] <-> COM Inputs/Data In 8
//     PlcTask Inputs/GVL_iXlinker.EtherCAT_Master_EPPxxxx.Beckhoff_EPP6xxx.Beckhoff_EPP6xxxEK1122.A_0001_EPP6001_0002_0016.COM_Inputs.Data_In[9] <-> COM Inputs/Data In 9
//     PlcTask Inputs/GVL_iXlinker.EtherCAT_Master_EPPxxxx.Beckhoff_EPP6xxx.Beckhoff_EPP6xxxEK1122.A_0001_EPP6001_0002_0016.COM_Inputs.Data_In[10] <-> COM Inputs/Data In 10
//     PlcTask Inputs/GVL_iXlinker.EtherCAT_Master_EPPxxxx.Beckhoff_EPP6xxx.Beckhoff_EPP6xxxEK1122.A_0001_EPP6001_0002_0016.COM_Inputs.Data_In[11] <-> COM Inputs/Data In 11
//     PlcTask Inputs/GVL_iXlinker.EtherCAT_Master_EPPxxxx.Beckhoff_EPP6xxx.Beckhoff_EPP6xxxEK1122.A_0001_EPP6001_0002_0016.COM_Inputs.Data_In[12] <-> COM Inputs/Data In 12
//     PlcTask Inputs/GVL_iXlinker.EtherCAT_Master_EPPxxxx.Beckhoff_EPP6xxx.Beckhoff_EPP6xxxEK1122.A_0001_EPP6001_0002_0016.COM_Inputs.Data_In[13] <-> COM Inputs/Data In 13
//     PlcTask Inputs/GVL_iXlinker.EtherCAT_Master_EPPxxxx.Beckhoff_EPP6xxx.Beckhoff_EPP6xxxEK1122.A_0001_EPP6001_0002_0016.COM_Inputs.Data_In[14] <-> COM Inputs/Data In 14
//     PlcTask Inputs/GVL_iXlinker.EtherCAT_Master_EPPxxxx.Beckhoff_EPP6xxx.Beckhoff_EPP6xxxEK1122.A_0001_EPP6001_0002_0016.COM_Inputs.Data_In[15] <-> COM Inputs/Data In 15
//     PlcTask Inputs/GVL_iXlinker.EtherCAT_Master_EPPxxxx.Beckhoff_EPP6xxx.Beckhoff_EPP6xxxEK1122.A_0001_EPP6001_0002_0016.COM_Inputs.Data_In[16] <-> COM Inputs/Data In 16
//     PlcTask Inputs/GVL_iXlinker.EtherCAT_Master_EPPxxxx.Beckhoff_EPP6xxx.Beckhoff_EPP6xxxEK1122.A_0001_EPP6001_0002_0016.COM_Inputs.Data_In[17] <-> COM Inputs/Data In 17
//     PlcTask Inputs/GVL_iXlinker.EtherCAT_Master_EPPxxxx.Beckhoff_EPP6xxx.Beckhoff_EPP6xxxEK1122.A_0001_EPP6001_0002_0016.COM_Inputs.Data_In[18] <-> COM Inputs/Data In 18
//     PlcTask Inputs/GVL_iXlinker.EtherCAT_Master_EPPxxxx.Beckhoff_EPP6xxx.Beckhoff_EPP6xxxEK1122.A_0001_EPP6001_0002_0016.COM_Inputs.Data_In[19] <-> COM Inputs/Data In 19
//     PlcTask Inputs/GVL_iXlinker.EtherCAT_Master_EPPxxxx.Beckhoff_EPP6xxx.Beckhoff_EPP6xxxEK1122.A_0001_EPP6001_0002_0016.COM_Inputs.Data_In[20] <-> COM Inputs/Data In 20
//     PlcTask Inputs/GVL_iXlinker.EtherCAT_Master_EPPxxxx.Beckhoff_EPP6xxx.Beckhoff_EPP6xxxEK1122.A_0001_EPP6001_0002_0016.COM_Inputs.Data_In[21] <-> COM Inputs/Data In 21
//     PlcTask Outputs/GVL_iXlinker.EtherCAT_Master_EPPxxxx.Beckhoff_EPP6xxx.Beckhoff_EPP6xxxEK1122.A_0001_EPP6001_0002_0016.COM_Outputs.Ctrl <-> COM Outputs/Ctrl
//     PlcTask Outputs/GVL_iXlinker.EtherCAT_Master_EPPxxxx.Beckhoff_EPP6xxx.Beckhoff_EPP6xxxEK1122.A_0001_EPP6001_0002_0016.COM_Outputs.Data_Out[0] <-> COM Outputs/Data Out 0
//     PlcTask Outputs/GVL_iXlinker.EtherCAT_Master_EPPxxxx.Beckhoff_EPP6xxx.Beckhoff_EPP6xxxEK1122.A_0001_EPP6001_0002_0016.COM_Outputs.Data_Out[1] <-> COM Outputs/Data Out 1
//     PlcTask Outputs/GVL_iXlinker.EtherCAT_Master_EPPxxxx.Beckhoff_EPP6xxx.Beckhoff_EPP6xxxEK1122.A_0001_EPP6001_0002_0016.COM_Outputs.Data_Out[2] <-> COM Outputs/Data Out 2
//     PlcTask Outputs/GVL_iXlinker.EtherCAT_Master_EPPxxxx.Beckhoff_EPP6xxx.Beckhoff_EPP6xxxEK1122.A_0001_EPP6001_0002_0016.COM_Outputs.Data_Out[3] <-> COM Outputs/Data Out 3
//     PlcTask Outputs/GVL_iXlinker.EtherCAT_Master_EPPxxxx.Beckhoff_EPP6xxx.Beckhoff_EPP6xxxEK1122.A_0001_EPP6001_0002_0016.COM_Outputs.Data_Out[4] <-> COM Outputs/Data Out 4
//     PlcTask Outputs/GVL_iXlinker.EtherCAT_Master_EPPxxxx.Beckhoff_EPP6xxx.Beckhoff_EPP6xxxEK1122.A_0001_EPP6001_0002_0016.COM_Outputs.Data_Out[5] <-> COM Outputs/Data Out 5
//     PlcTask Outputs/GVL_iXlinker.EtherCAT_Master_EPPxxxx.Beckhoff_EPP6xxx.Beckhoff_EPP6xxxEK1122.A_0001_EPP6001_0002_0016.COM_Outputs.Data_Out[6] <-> COM Outputs/Data Out 6
//     PlcTask Outputs/GVL_iXlinker.EtherCAT_Master_EPPxxxx.Beckhoff_EPP6xxx.Beckhoff_EPP6xxxEK1122.A_0001_EPP6001_0002_0016.COM_Outputs.Data_Out[7] <-> COM Outputs/Data Out 7
//     PlcTask Outputs/GVL_iXlinker.EtherCAT_Master_EPPxxxx.Beckhoff_EPP6xxx.Beckhoff_EPP6xxxEK1122.A_0001_EPP6001_0002_0016.COM_Outputs.Data_Out[8] <-> COM Outputs/Data Out 8
//     PlcTask Outputs/GVL_iXlinker.EtherCAT_Master_EPPxxxx.Beckhoff_EPP6xxx.Beckhoff_EPP6xxxEK1122.A_0001_EPP6001_0002_0016.COM_Outputs.Data_Out[9] <-> COM Outputs/Data Out 9
//     PlcTask Outputs/GVL_iXlinker.EtherCAT_Master_EPPxxxx.Beckhoff_EPP6xxx.Beckhoff_EPP6xxxEK1122.A_0001_EPP6001_0002_0016.COM_Outputs.Data_Out[10] <-> COM Outputs/Data Out 10
//     PlcTask Outputs/GVL_iXlinker.EtherCAT_Master_EPPxxxx.Beckhoff_EPP6xxx.Beckhoff_EPP6xxxEK1122.A_0001_EPP6001_0002_0016.COM_Outputs.Data_Out[11] <-> COM Outputs/Data Out 11
//     PlcTask Outputs/GVL_iXlinker.EtherCAT_Master_EPPxxxx.Beckhoff_EPP6xxx.Beckhoff_EPP6xxxEK1122.A_0001_EPP6001_0002_0016.COM_Outputs.Data_Out[12] <-> COM Outputs/Data Out 12
//     PlcTask Outputs/GVL_iXlinker.EtherCAT_Master_EPPxxxx.Beckhoff_EPP6xxx.Beckhoff_EPP6xxxEK1122.A_0001_EPP6001_0002_0016.COM_Outputs.Data_Out[13] <-> COM Outputs/Data Out 13
//     PlcTask Outputs/GVL_iXlinker.EtherCAT_Master_EPPxxxx.Beckhoff_EPP6xxx.Beckhoff_EPP6xxxEK1122.A_0001_EPP6001_0002_0016.COM_Outputs.Data_Out[14] <-> COM Outputs/Data Out 14
//     PlcTask Outputs/GVL_iXlinker.EtherCAT_Master_EPPxxxx.Beckhoff_EPP6xxx.Beckhoff_EPP6xxxEK1122.A_0001_EPP6001_0002_0016.COM_Outputs.Data_Out[15] <-> COM Outputs/Data Out 15
//     PlcTask Outputs/GVL_iXlinker.EtherCAT_Master_EPPxxxx.Beckhoff_EPP6xxx.Beckhoff_EPP6xxxEK1122.A_0001_EPP6001_0002_0016.COM_Outputs.Data_Out[16] <-> COM Outputs/Data Out 16
//     PlcTask Outputs/GVL_iXlinker.EtherCAT_Master_EPPxxxx.Beckhoff_EPP6xxx.Beckhoff_EPP6xxxEK1122.A_0001_EPP6001_0002_0016.COM_Outputs.Data_Out[17] <-> COM Outputs/Data Out 17
//     PlcTask Outputs/GVL_iXlinker.EtherCAT_Master_EPPxxxx.Beckhoff_EPP6xxx.Beckhoff_EPP6xxxEK1122.A_0001_EPP6001_0002_0016.COM_Outputs.Data_Out[18] <-> COM Outputs/Data Out 18
//     PlcTask Outputs/GVL_iXlinker.EtherCAT_Master_EPPxxxx.Beckhoff_EPP6xxx.Beckhoff_EPP6xxxEK1122.A_0001_EPP6001_0002_0016.COM_Outputs.Data_Out[19] <-> COM Outputs/Data Out 19
//     PlcTask Outputs/GVL_iXlinker.EtherCAT_Master_EPPxxxx.Beckhoff_EPP6xxx.Beckhoff_EPP6xxxEK1122.A_0001_EPP6001_0002_0016.COM_Outputs.Data_Out[20] <-> COM Outputs/Data Out 20
//     PlcTask Outputs/GVL_iXlinker.EtherCAT_Master_EPPxxxx.Beckhoff_EPP6xxx.Beckhoff_EPP6xxxEK1122.A_0001_EPP6001_0002_0016.COM_Outputs.Data_Out[21] <-> COM Outputs/Data Out 21
//     PlcTask Inputs/GVL_iXlinker.EtherCAT_Master_EPPxxxx.Beckhoff_EPP6xxx.Beckhoff_EPP6xxxEK1122.A_0001_EPP6001_0002_0016.WcState.WcState <-> WcState/WcState
//     PlcTask Inputs/GVL_iXlinker.EtherCAT_Master_EPPxxxx.Beckhoff_EPP6xxx.Beckhoff_EPP6xxxEK1122.A_0001_EPP6001_0002_0016.WcState.InputToggle <-> WcState/InputToggle
//     PlcTask Inputs/GVL_iXlinker.EtherCAT_Master_EPPxxxx.Beckhoff_EPP6xxx.Beckhoff_EPP6xxxEK1122.A_0001_EPP6001_0002_0016.InfoData.AdsAddr <-> InfoData/AdsAddr
//     PlcTask Inputs/GVL_iXlinker.EtherCAT_Master_EPPxxxx.Beckhoff_EPP6xxx.Beckhoff_EPP6xxxEK1122.A_0001_EPP6001_0002_0016.InfoData.State <-> InfoData/State
//   PLC/PLC Instance <-> EtherCAT Master EPPxxxx/Beckhoff EPP6xxx/Beckhoff EPP6xxxEK1122/A_0002(EPP6001-0002-0017)
//     PlcTask Inputs/GVL_iXlinker.EtherCAT_Master_EPPxxxx.Beckhoff_EPP6xxx.Beckhoff_EPP6xxxEK1122.A_0002_EPP6001_0002_0017.COM_Inputs.Status <-> COM Inputs/Status
//     PlcTask Inputs/GVL_iXlinker.EtherCAT_Master_EPPxxxx.Beckhoff_EPP6xxx.Beckhoff_EPP6xxxEK1122.A_0002_EPP6001_0002_0017.COM_Inputs.Data_In[0] <-> COM Inputs/Data In 0
//     PlcTask Inputs/GVL_iXlinker.EtherCAT_Master_EPPxxxx.Beckhoff_EPP6xxx.Beckhoff_EPP6xxxEK1122.A_0002_EPP6001_0002_0017.COM_Inputs.Data_In[1] <-> COM Inputs/Data In 1
//     PlcTask Inputs/GVL_iXlinker.EtherCAT_Master_EPPxxxx.Beckhoff_EPP6xxx.Beckhoff_EPP6xxxEK1122.A_0002_EPP6001_0002_0017.COM_Inputs.Data_In[2] <-> COM Inputs/Data In 2
//     PlcTask Inputs/GVL_iXlinker.EtherCAT_Master_EPPxxxx.Beckhoff_EPP6xxx.Beckhoff_EPP6xxxEK1122.A_0002_EPP6001_0002_0017.COM_Inputs.Data_In[3] <-> COM Inputs/Data In 3
//     PlcTask Inputs/GVL_iXlinker.EtherCAT_Master_EPPxxxx.Beckhoff_EPP6xxx.Beckhoff_EPP6xxxEK1122.A_0002_EPP6001_0002_0017.COM_Inputs.Data_In[4] <-> COM Inputs/Data In 4
//     PlcTask Inputs/GVL_iXlinker.EtherCAT_Master_EPPxxxx.Beckhoff_EPP6xxx.Beckhoff_EPP6xxxEK1122.A_0002_EPP6001_0002_0017.COM_Inputs.Data_In[5] <-> COM Inputs/Data In 5
//     PlcTask Inputs/GVL_iXlinker.EtherCAT_Master_EPPxxxx.Beckhoff_EPP6xxx.Beckhoff_EPP6xxxEK1122.A_0002_EPP6001_0002_0017.COM_Inputs.Data_In[6] <-> COM Inputs/Data In 6
//     PlcTask Inputs/GVL_iXlinker.EtherCAT_Master_EPPxxxx.Beckhoff_EPP6xxx.Beckhoff_EPP6xxxEK1122.A_0002_EPP6001_0002_0017.COM_Inputs.Data_In[7] <-> COM Inputs/Data In 7
//     PlcTask Inputs/GVL_iXlinker.EtherCAT_Master_EPPxxxx.Beckhoff_EPP6xxx.Beckhoff_EPP6xxxEK1122.A_0002_EPP6001_0002_0017.COM_Inputs.Data_In[8] <-> COM Inputs/Data In 8
//     PlcTask Inputs/GVL_iXlinker.EtherCAT_Master_EPPxxxx.Beckhoff_EPP6xxx.Beckhoff_EPP6xxxEK1122.A_0002_EPP6001_0002_0017.COM_Inputs.Data_In[9] <-> COM Inputs/Data In 9
//     PlcTask Inputs/GVL_iXlinker.EtherCAT_Master_EPPxxxx.Beckhoff_EPP6xxx.Beckhoff_EPP6xxxEK1122.A_0002_EPP6001_0002_0017.COM_Inputs.Data_In[10] <-> COM Inputs/Data In 10
